(* CoDeSys 2.3.9.13 project: wago_842_1.8.pro *)
(* Libraries: X:\Dev\Wago Calaos\Wago_1.7\DALI_02v2.4.lib 10.3.09 10:32:26, SYSTEM.LIB 6.12.00 08:50:26, Visual.lib 22.2.01 17:57:44, mod_com.lib 17.5.05 08:45:02, Ethernet.lib 8.7.04 10:03:04, Standard.lib 1.12.04 09:59:26 *)

(* PLC configuration (modules and I/O channels)
K-Bus [K_Bus] node 0, in %IB0 out %QB0
Fieldbus variables [FB_VARS] node 1, in %IB512 out %QB512
*)

(* Global variable list: Variables_Globales *)
VAR_GLOBAL
	ConfigDone: BOOL := FALSE; (* Do the config only one time *)
	info : ARRAY[0..63] OF MODULE_INFO; (* I/O Module infos *)

	(* modules infos *)
	nb_module: BYTE;
	nb_module_in: BYTE;
	nb_module_out: BYTE;
	nb_module_analog_in: BYTE;
	nb_module_analog_out: BYTE;
	start_addr_in: WORD;
	start_addr_out: WORD;
	nb_input_digital: WORD;
	nb_output_digital: WORD;

	(* All inputs events *)
	event: ARRAY[0..200] OF INTER_EVENT; (* MAX of 256/8 = 32 digital input modules *)
	lights: ARRAY[0..31] OF BYTE;	(* MAX of 256/8 = 32 digital output modules as lights *)
									(* We store only the boolean state of each light *)
	volets: ARRAY[0..100] OF VOLET; (* MAX of 256/8 = 32 digital output modules as volets *)

	HEARTBEAT: BOOL := FALSE;

	OutArrState: ARRAY[0..512] OF BYTE;	(* state of outputs *)

	impulse_time: TIME := T#300ms;

	(* DALI *)
	DALIJoblist: FbDALI_Joblist;

	Dali_switch: FbDALI_SwitchValue;
	DALIDimmValue: FbDALI_StatusDimmValue;

	byOutArr AT %QB0: ARRAY[0..512] OF BYTE;	(* Byte array in Q memory *)
	byInArr AT %IB0: ARRAY[0..512] OF BYTE;	(* Byte array in I memory *)
END_VAR

(* Data type *)
TYPE OUTPUT_ADDR :
STRUCT

	(* the first ouput address, only needed *)
	ADDR1: BYTE;
	(* the second address used only for the VOLET function bloc *)
	ADDR2: BYTE;

	(* If SameAs <> -1, then a input is wired the same as the specified ID *)
	SameAs: INT := -1;

END_STRUCT
END_TYPE

(* Data type *)
(* Enumerate all type of output.
	NONE: Do nothing.
	TELERUPTEUR: Simulate a telerupteur.
	DIRECT: The input is directly "wired" to the output.
	VOLET: Simulate a volet with one button and 2 output (up and down).
	TELERUPTEUR_DALI: Controls a DALI lamp
	TELERUPTEUR_DALI_GROUP: Controls a DALI group
*)

TYPE OUTPUT_TYPE : (NONE, TELERUPTEUR, DIRECT, VOLET, VOLET_IMPULSE, TELERUPTEUR_DALI, TELERUPTEUR_DALI_GROUP);
END_TYPE

(* Data type *)
(* Enumerate all type of output.
	NONE: Do nothing.
	TELERUPTEUR: Simulate a telerupteur.
	DIRECT: The input is directly "wired" to the output.
	VOLET: Simulate a volet with one button and 2 output (up and down).
*)

TYPE VOLET_MODE : (VOLET_STOP, VOLET_UP, VOLET_DOWN, IMP_UP, IMP_DOWN, IMP_STOP);
END_TYPE

(* POU PLC_PRG, ST *)
PROGRAM PLC_PRG
VAR
	i: INT;
	start: BYTE;
	init_dali: BOOL := FALSE;
END_VAR
(* Main PRG *)

(* Start the config program *)
Config;

IF (Config.CONFIG_DALI = TRUE) THEN

	(* Call DALI jobs to send commands on the DALI bus *)
	DALIJoblist();
	DALI_Config();

	IF (init_dali = FALSE) THEN
		Dali_switch(xButton := FALSE);
		Dali_switch(bAddress := 255, xGroup := FALSE, bDimmLevel := 0,
				         xButton := TRUE);

		init_dali := TRUE;
	END_IF

END_IF


IF (HEARTBEAT = FALSE) THEN
	ManageOutput;
END_IF

(* Read a command from UDP *)
UDPServer;

(* Send inputs status on the network *)
SendInput;

IF (HEARTBEAT = FALSE) THEN
	(* update outputs *)
	FOR i := start_addr_out / 8 TO 512 DO
		byOutArr[i] := OutArrState[i];
	END_FOR
ELSE
	(* update outputs *)
	FOR i := start_addr_out / 8 TO 512 DO
		OutArrState[i] := byOutArr[i];
	END_FOR
END_IF
END_PROGRAM

(* POU Config, ST *)
PROGRAM Config
VAR
	access : MODULE_INFO_ACCESS;
	cpt: BYTE;
	ethernet_config : ETHERNET_SET_VARIABLES;
	CONFIG_DALI: BOOL;

END_VAR
VAR_INPUT RETAIN
	SERVER_IP: DWORD;
	DALI_MODE: BYTE;
END_VAR
VAR CONSTANT
	CALAOS_VERSION_H: WORD := 1;
	CALAOS_VERSION_L: WORD := 8;
	DALI: BYTE := 1;
	DSI: BYTE := 2;
END_VAR
(* Do all the config job *)

IF (ConfigDone = FALSE) THEN

(* Get the module I/O Config *)
access.physicalPosTo := 0;
access.moduleType := 0;
ADD_PI_INFORMATION( 1, ADR(access), ADR(info[0]) );

FOR cpt := 0 TO 63 DO
	IF (info[cpt].moduleType = 0 AND info[cpt].physicalPos = 0) THEN
		cpt := 63; (* the end *)
	ELSE
		IF (info[cpt].moduleType = 641) THEN
			(* This is a DALI module *)
			CONFIG_DALI := TRUE;
		END_IF

		nb_module := nb_module + 1;
		IF ((info[cpt].desc.sizePAE > 8) AND (info[cpt].desc.channels > 0)) THEN
			nb_module_analog_in := nb_module_analog_in + 1;
			start_addr_in := start_addr_in + info[cpt].desc.sizePAE;
		END_IF
		IF ((info[cpt].desc.sizePAA > 8) AND (info[cpt].desc.channels > 0)) THEN
			nb_module_analog_out := nb_module_analog_out + 1;
			start_addr_out := start_addr_out + info[cpt].desc.sizePAA;
		END_IF
		IF ((info[cpt].desc.sizePAE <= 16) AND (info[cpt].desc.sizePAE > 0) AND (info[cpt].desc.channels = 0)) THEN
			nb_module_in := nb_module_in + 1;
			nb_input_digital := nb_input_digital + info[cpt].desc.sizePAE;
		END_IF
		IF ((info[cpt].desc.sizePAA <= 16) AND (info[cpt].desc.sizePAA > 0) AND (info[cpt].desc.channels = 0)) THEN
			nb_module_out := nb_module_out + 1;
			nb_output_digital := nb_output_digital + info[cpt].desc.sizePAA;
		END_IF

	END_IF
END_FOR

(* Start the heartbeat timer *)
(*HEARTBEAT_TIMER(IN:=FALSE, PT:=T#30s);*)
(*HEARTBEAT_TIMER(IN:=TRUE, PT:=T#30s);*)

(* Config du timout des sockets *)
ethernet_config(EN:=TRUE, BootpRequest:=0, ConnectionWdTime:=65535);

ConfigDone := TRUE;

LedInit;
LedStart;

END_IF
END_PROGRAM

(* POU LedInit, ST *)
PROGRAM LedInit
VAR
	Sequence: ARRAY [0..4] OF FLASHING_SEQUENCE;
	ptrFS: POINTER TO FLASHING_SEQUENCE;

END_VAR
Sequence[0].Colour := ORANGE;
Sequence[0].Frequency := 10;
Sequence[0].Relation := 50;
Sequence[0].Duration := t#0s;

Sequence[1].Colour := ORANGE;
Sequence[1].Frequency := 0;
Sequence[1].Relation := 128;
Sequence[1].Duration := t#0s;

Sequence[2].Colour := GREEN;
Sequence[2].Frequency := 0;
Sequence[2].Relation := 128;
Sequence[2].Duration := t#0s;

Sequence[3].Colour := RED;
Sequence[3].Frequency := 0;
Sequence[3].Relation := 128;
Sequence[3].Duration := t#0s;

Sequence[4].Colour := ORANGE;
Sequence[4].Frequency := 0;
Sequence[4].Relation := 0;
Sequence[4].Duration := t#0s;

ptrFS := ADR(Sequence);
SET_FLASHING_SEQUENCE(TRUE, ADR(ptrFS));
END_PROGRAM

(* POU LedStart, ST *)
PROGRAM LedStart
VAR
END_VAR
SET_FLASHING_SEQUENCE_INDEX(TRUE, TRUE, 0);
START_FLASHING_SEQUENCE(TRUE);
END_PROGRAM

(* POU ManageOutput, ST *)
PROGRAM ManageOutput
VAR
	cpt: BYTE;
	tmp: BYTE;
	_light: LIGHT;
END_VAR
VAR_INPUT RETAIN
	output_type: ARRAY[0..256] OF OUTPUT_TYPE; (* The type of each output *)
	output_addr: ARRAY[0..256] OF OUTPUT_ADDR; (* The addresses for each type *)
    	volets_position: ARRAY[0..30] OF DWORD;
END_VAR
(* Set all outputs when in standalone mode *)

(* Get the address of the first digital output *)
FOR cpt := 0 TO UINT_TO_BYTE(nb_input_digital) DO

	CASE output_type[cpt] OF
	NONE: (* Do nothing *);
	TELERUPTEUR:
		tmp := cpt;
		IF (output_addr[cpt].SameAs >= 0) THEN
			tmp := INT_TO_BYTE(output_addr[cpt].SameAs);
		END_IF
		IF (event[cpt].ON = TRUE) THEN
			_light(IN := FALSE, STATE := BYTE_TO_BOOL(SHR(lights[tmp / 8], tmp MOD 8) AND 16#01));
			_light(IN := TRUE, STATE := BYTE_TO_BOOL(SHR(lights[tmp / 8], tmp MOD 8) AND 16#01));
			SetOutput(output_addr[tmp].ADDR1 + start_addr_out, _light.OUT);

			(* set old state *)
			IF (_light.OUT = TRUE) THEN
				lights[tmp / 8] := lights[tmp / 8] OR SHL(16#01, tmp MOD 8);
			ELSE
				lights[tmp / 8] := lights[tmp / 8] AND NOT SHL(16#01, tmp MOD 8);
			END_IF
		END_IF
	DIRECT:
		tmp := cpt;
		IF (output_addr[cpt].SameAs >= 0) THEN
			tmp := INT_TO_BYTE(output_addr[cpt].SameAs);
		END_IF
		SetOutput(output_addr[tmp].ADDR1 + start_addr_out, GetInput(cpt + start_addr_in));
	VOLET:
		tmp := cpt;
		IF (output_addr[cpt].SameAs >= 0) THEN
			tmp := INT_TO_BYTE(output_addr[cpt].SameAs);
		END_IF
		IF (event[cpt].ON = TRUE) THEN
			volets[tmp](IN := TRUE, IMPULSE := FALSE);
			SetOutput(output_addr[tmp].ADDR1 + start_addr_out, volets[tmp].MONTE);
			SetOutput(output_addr[tmp].ADDR2 + start_addr_out, volets[tmp].DESCENTE);
		END_IF
	VOLET_IMPULSE:
		tmp := cpt;
		IF (output_addr[cpt].SameAs >= 0) THEN
			tmp := INT_TO_BYTE(output_addr[cpt].SameAs);
		END_IF
		IF (event[cpt].ON = TRUE) THEN
			volets[tmp](IN := TRUE, IMPULSE := TRUE);
		ELSE
			volets[tmp](IN := FALSE, IMPULSE := TRUE);
		END_IF
		SetOutput(output_addr[tmp].ADDR1 + start_addr_out, volets[tmp].MONTE);
		SetOutput(output_addr[tmp].ADDR2 + start_addr_out, volets[tmp].DESCENTE);
	TELERUPTEUR_DALI:
		tmp := cpt;
		IF (output_addr[cpt].SameAs >= 0) THEN
			tmp := INT_TO_BYTE(output_addr[cpt].SameAs);
		END_IF
		IF (event[cpt].ON = TRUE) THEN
			_light(IN := FALSE, STATE := BYTE_TO_BOOL(SHR(lights[tmp / 8], tmp MOD 8) AND 16#01));
			_light(IN := TRUE, STATE := BYTE_TO_BOOL(SHR(lights[tmp / 8], tmp MOD 8) AND 16#01));

			Dali_switch(xButton := FALSE);
			IF (_light.OUT = TRUE) THEN
				Dali_switch(bAddress := output_addr[tmp].ADDR2, xGroup := FALSE, bDimmLevel := 100,
					bFadeTime := 1, xButton := TRUE);
			ELSE
				Dali_switch(bAddress := output_addr[tmp].ADDR2, xGroup := FALSE, bDimmLevel := 0,
					bFadeTime := 1, xButton := TRUE);
			END_IF

			(* set old state *)
			IF (_light.OUT = TRUE) THEN
				lights[tmp / 8] := lights[tmp / 8] OR SHL(16#01, tmp MOD 8);
			ELSE
				lights[tmp / 8] := lights[tmp / 8] AND NOT SHL(16#01, tmp MOD 8);
			END_IF
		END_IF
	TELERUPTEUR_DALI_GROUP:
		tmp := cpt;
		IF (output_addr[cpt].SameAs >= 0) THEN
			tmp := INT_TO_BYTE(output_addr[cpt].SameAs);
		END_IF
		IF (event[cpt].ON = TRUE) THEN
			_light(IN := FALSE, STATE := BYTE_TO_BOOL(SHR(lights[tmp / 8], tmp MOD 8) AND 16#01));
			_light(IN := TRUE, STATE := BYTE_TO_BOOL(SHR(lights[tmp / 8], tmp MOD 8) AND 16#01));
			Dali_switch(xButton := FALSE);
			IF (_light.OUT = TRUE) THEN
				Dali_switch(bAddress := output_addr[tmp].ADDR2, xGroup := TRUE, bDimmLevel := 100,
					bFadeTime := 1, xButton := TRUE);
			ELSE
				Dali_switch(bAddress := output_addr[tmp].ADDR2, xGroup := TRUE, bDimmLevel := 0,
					bFadeTime := 1, xButton := TRUE);
			END_IF

			(* set old state *)
			IF (_light.OUT = TRUE) THEN
				lights[tmp / 8] := lights[tmp / 8] OR SHL(16#01, tmp MOD 8);
			ELSE
				lights[tmp / 8] := lights[tmp / 8] AND NOT SHL(16#01, tmp MOD 8);
			END_IF
		END_IF
	END_CASE
END_FOR
END_PROGRAM

(* POU LIGHT, ST *)
FUNCTION_BLOCK LIGHT
VAR
	TRIG: R_TRIG;
	light: BOOL;
END_VAR
VAR_INPUT
	IN: BOOL;
	STATE: BOOL;
END_VAR
VAR_OUTPUT
	OUT: BOOL;
END_VAR
(* telerupteur *)

TRIG(CLK := IN);
light := TRIG.Q;

OUT := STATE;

IF light = TRUE THEN
	IF OUT = TRUE THEN
		OUT := FALSE;
	ELSE
		OUT := TRUE;
	END_IF;
END_IF;
END_FUNCTION_BLOCK

(* POU SetOutput, ST *)
FUNCTION SetOutput : BOOL
VAR_INPUT
	bit_offset: UINT;
	val: BOOL;
END_VAR
VAR
END_VAR
(* get the byte AND  select the bit *)

(* Take care of special modules *
bit_offset := bit_offset + start_addr_out; *)

IF (HEARTBEAT = FALSE) THEN
	IF (val = TRUE) THEN
		OutArrState[bit_offset / 8] := OutArrState[bit_offset / 8] OR SHL(16#01, bit_offset MOD 8);
	ELSE
		OutArrState[bit_offset / 8] := OutArrState[bit_offset / 8] AND NOT SHL(16#01, bit_offset MOD 8);
	END_IF

ELSE
	IF (val = TRUE) THEN
		byOutArr[bit_offset / 8] := byOutArr[bit_offset / 8] OR SHL(16#01, bit_offset MOD 8);
	ELSE
		byOutArr[bit_offset / 8] := byOutArr[bit_offset / 8] AND NOT SHL(16#01, bit_offset MOD 8);
	END_IF
END_IF

SetOutput := TRUE;
END_FUNCTION

(* POU GetInput, ST *)
FUNCTION GetInput : BOOL
VAR_INPUT
	bit_offset: UINT;
END_VAR
VAR
END_VAR
VAR CONSTANT
	byBitArr: ARRAY[0..7] OF BYTE := 16#01,16#02,16#04,16#08,16#10,16#20,16#40,16#80;
END_VAR
(* get the byte AND  select the bit *)

GetInput := BYTE_TO_BOOL(byInArr[bit_offset/8] AND byBitArr[bit_offset MOD 8]);
END_FUNCTION

(* POU VOLET, ST *)
FUNCTION_BLOCK VOLET
VAR
	sens: BOOL;
	imp: TP;
	mode: VOLET_MODE;
END_VAR
VAR_INPUT
	IN: BOOL;
	IMPULSE: BOOL;
END_VAR
VAR_OUTPUT
	MONTE: BOOL;
	DESCENTE:BOOL;
END_VAR
(* Volet *)

IF IMPULSE = FALSE THEN
	(* Normal mode *)
	IF (MONTE = TRUE OR DESCENTE = TRUE) THEN
		MONTE := FALSE;
		DESCENTE := FALSE;
	ELSE

		IF IN = TRUE THEN
			IF sens = TRUE THEN
				sens := FALSE;
			ELSE
				sens := TRUE;
			END_IF;

			IF sens = TRUE THEN
				(*monte*)
				DESCENTE := FALSE;
				MONTE := TRUE;
			ELSE
				MONTE := FALSE;
				DESCENTE := TRUE;
			END_IF;
		END_IF

	END_IF
ELSE
	(* impulse mode *)
	imp(IN := FALSE, PT:= impulse_time);

	IF mode = IMP_STOP THEN
		MONTE := imp.Q;
		DESCENTE := imp.Q;
		IF imp.Q = FALSE THEN
			mode := VOLET_STOP;
		END_IF;
	END_IF;
	IF mode = IMP_UP THEN
		MONTE := imp.Q;
		DESCENTE := FALSE;
		IF imp.Q = FALSE THEN
			mode := VOLET_UP;
		END_IF;
	END_IF;
	IF mode = IMP_DOWN THEN
		MONTE := FALSE;
		DESCENTE := imp.Q;
		IF imp.Q = FALSE THEN
			mode := VOLET_DOWN;
		END_IF;
	END_IF;

	IF mode = VOLET_UP OR mode = VOLET_DOWN THEN
		IF IN = TRUE THEN
			imp(IN := TRUE, PT:= impulse_time);
			mode := IMP_STOP;
		END_IF;
	ELSE
		IF IN = TRUE THEN
			IF sens = TRUE THEN
				sens := FALSE;
			ELSE
				sens := TRUE;
			END_IF;

			IF sens = TRUE THEN
				imp(IN := TRUE, PT:= impulse_time);
				mode := IMP_UP;
			ELSE
				imp(IN := TRUE, PT:= impulse_time);
				mode := IMP_DOWN;
			END_IF;
		END_IF;
	END_IF;
END_IF;
END_FUNCTION_BLOCK

(* POU UDPServer, ST *)
PROGRAM UDPServer
VAR
	server: EthernetServer_FB;

	rBuffer, wBuffer: POINTER TO BYTE;
	buffer: ARRAY[1 .. 1500] OF BYTE;
	cmd: STRING(255);
	start_send: BOOL := FALSE;
	i: WORD;
	dali_group: BOOL;

	HEARTBEAT_TIMER: TON;

	p1: DINT;
	p2: DINT;
	p3: DINT;
	p4: DINT;
	p5: DINT;
	ip1, ip2, ip3, ip4: DWORD;
	DaliSend: BOOL := FALSE;

	(* Used by dali config for answer
	   0 = no action
	   1 = Search all active address
	   2 = Read groups for short adress
	*)
	DaliSendAction: BYTE := 0;

(*	DALIShowShortAdr: FbDALI_ShowShortAdr;
	DALIConfigDevice: FbDALI_ConfigDevice;*)

END_VAR
(* Here we start an UDP server for other network functions *)

HEARTBEAT_TIMER(IN:=TRUE, PT:=T#30s);

rBuffer := ADR(buffer);
wBuffer := ADR(cmd);

cmd := CONCAT(cmd, ASCIIBYTE_TO_STRING(0));

server.tTIMEOUT	:= t#60s;
server.xTCP_PROTOCOL := FALSE;
server.wPORT := 4646;
server.iBYTES_TO_SEND := LEN(cmd) + 1;
server(xOPEN_SERVER := TRUE, xSTART_SEND := start_send, ptSEND_BUFFER := wBuffer, ptRECV_BUFFER := rBuffer);

IF server.bDataReceived THEN

	cmd := '';
	FOR i := 1 TO server.iBYTES_RECEIVED DO
		cmd := CONCAT(cmd, ASCIIBYTE_TO_STRING(buffer[i]));
	END_FOR

	IF (STRING_COMPARE(cmd, 'WAGO_HEARTBEAT') = TRUE) THEN
		HEARTBEAT_TIMER(IN:=FALSE, PT:=T#30s);
		HEARTBEAT_TIMER(IN:=TRUE, PT:=T#30s);

		LedModePC;
	END_IF

	IF (Strncmp(cmd, 'WAGO_SET_OUTTYPE ', 17) = TRUE) THEN
		p1 := GET_PARAM_DINT(cmd, 1);
		p2 := GET_PARAM_DINT(cmd, 2);
		CASE p2 OF
		0: ManageOutput.output_type[p1] := NONE;
		1: ManageOutput.output_type[p1] := TELERUPTEUR;
		2: ManageOutput.output_type[p1] := DIRECT;
		3: ManageOutput.output_type[p1] := VOLET;
		4: ManageOutput.output_type[p1] := VOLET_IMPULSE;
		5: ManageOutput.output_type[p1] := TELERUPTEUR_DALI;
		6: ManageOutput.output_type[p1] := TELERUPTEUR_DALI_GROUP;
		END_CASE
	END_IF

	IF (Strncmp(cmd, 'WAGO_SET_OUTADDR ', 17) = TRUE) THEN
		p1 := GET_PARAM_DINT(cmd, 1);
		p2 := GET_PARAM_DINT(cmd, 2);
		p3 := GET_PARAM_DINT(cmd, 3);
		p4 := GET_PARAM_DINT(cmd, 4);
		ManageOutput.output_addr[p1].ADDR1 := DINT_TO_BYTE(p2);
		ManageOutput.output_addr[p1].ADDR2 := DINT_TO_BYTE(p3);
		ManageOutput.output_addr[p1].SameAs := DINT_TO_INT(p4);
	END_IF

	IF (Strncmp(cmd, 'WAGO_GET_OUTTYPE ', 17) = TRUE) THEN
		p1 := GET_PARAM_DINT(cmd, 1);
		cmd := 'WAGO_OUTTYPE ';
		cmd := CONCAT(cmd, ITOA(DINT_TO_INT(p1)));
		cmd := CONCAT(cmd, ' ');
		CASE ManageOutput.output_type[p1] OF
		NONE: cmd := CONCAT(cmd, ITOA(0));;
		TELERUPTEUR: cmd := CONCAT(cmd, ITOA(1));;
		DIRECT: cmd := CONCAT(cmd, ITOA(2));;
		VOLET: cmd := CONCAT(cmd, ITOA(3));;
		VOLET_IMPULSE: cmd := CONCAT(cmd, ITOA(4));;
		TELERUPTEUR_DALI: cmd := CONCAT(cmd, ITOA(5));;
		TELERUPTEUR_DALI_GROUP: cmd := CONCAT(cmd, ITOA(6));;
		END_CASE
		start_send := TRUE;
	END_IF

	IF (Strncmp(cmd, 'WAGO_GET_OUTADDR ', 17) = TRUE) THEN
		p1 := GET_PARAM_DINT(cmd, 1);
		cmd := 'WAGO_OUTADDR ';
		cmd := CONCAT(cmd, ITOA(DINT_TO_INT(p1)));
		cmd := CONCAT(cmd, ' ');
		cmd := CONCAT(cmd, ITOA(ManageOutput.output_addr[p1].ADDR1));
		cmd := CONCAT(cmd, ' ');
		cmd := CONCAT(cmd, ITOA(ManageOutput.output_addr[p1].ADDR2));
		cmd := CONCAT(cmd, ' ');
		cmd := CONCAT(cmd, ITOA(ManageOutput.output_addr[p1].SameAs));
		start_send := TRUE;
	END_IF

	IF (STRING_COMPARE(cmd, 'WAGO_GET_INFO') = TRUE) THEN
		cmd := 'WAGO_INFO ';
		cmd := CONCAT(cmd, ITOA(nb_module));
		cmd := CONCAT(cmd, ' ');
		cmd := CONCAT(cmd, ITOA(nb_module_in));
		cmd := CONCAT(cmd, ' ');
		cmd := CONCAT(cmd, ITOA(WORD_TO_INT(nb_module_out)));
		cmd := CONCAT(cmd, ' ');
		cmd := CONCAT(cmd, ITOA(WORD_TO_INT(nb_input_digital)));
		cmd := CONCAT(cmd, ' ');
		cmd := CONCAT(cmd, ITOA(WORD_TO_INT(nb_output_digital)));
		cmd := CONCAT(cmd, ' ');
		cmd := CONCAT(cmd, ITOA(nb_module_analog_in));
		cmd := CONCAT(cmd, ' ');
		cmd := CONCAT(cmd, ITOA(nb_module_analog_out));
		start_send := TRUE;
	END_IF

	IF (Strncmp(cmd, 'WAGO_GET_INFO_MODULE ', 21) = TRUE) THEN
		p1 := GET_PARAM_DINT(cmd, 1);
		cmd := 'WAGO_MODULE ';
		cmd := CONCAT(cmd, ITOA(DINT_TO_INT(p1)));
		cmd := CONCAT(cmd, ' ');
		cmd := CONCAT(cmd, ITOA(WORD_TO_INT(info[p1].moduleType)));
		cmd := CONCAT(cmd, ' ');
		cmd := CONCAT(cmd, ITOA(info[p1].physicalPos));
		cmd := CONCAT(cmd, ' ');
		cmd := CONCAT(cmd, ITOA(info[p1].desc.sizePAE));
		cmd := CONCAT(cmd, ' ');
		cmd := CONCAT(cmd, ITOA(info[p1].desc.sizePAA));
		start_send := TRUE;
	END_IF

	IF (Strncmp(cmd, 'WAGO_SET_SERVER_IP ', 19) = TRUE) THEN
		cmd := DELETE(cmd, 19, 1);
		(* deletes the dot  *)
		cmd := REPLACE(cmd, ' ', 1, FIND(cmd, '.'));
		cmd := REPLACE(cmd, ' ', 1, FIND(cmd, '.'));
		cmd := REPLACE(cmd, ' ', 1, FIND(cmd, '.'));
		ip1 := GET_PARAM_DINT(cmd, 0);
		ip2 := GET_PARAM_DINT(cmd, 1);
		ip3 := GET_PARAM_DINT(cmd, 2);
		ip4 := GET_PARAM_DINT(cmd, 3);
		Config.SERVER_IP := SHL(ip1, 24) OR SHL(ip2, 16) OR SHL(ip3, 8) OR ip4;
	END_IF

	IF (Strncmp(cmd, 'WAGO_SET_OUTPUT ', 16) = TRUE) THEN
		p1 := GET_PARAM_DINT(cmd, 1);
		p2 := GET_PARAM_DINT(cmd, 2);

		p1 := start_addr_out + p1;

		IF (p2 = 1) THEN
			SetOutput(DINT_TO_UINT(p1), TRUE);
		ELSE
			SetOutput(DINT_TO_UINT(p1), FALSE);
		END_IF
	END_IF

	IF (Strncmp(cmd, 'WAGO_GET_VERSION', 16) = TRUE) THEN
		cmd := 'WAGO_GET_VERSION ';
		cmd := CONCAT(cmd, ITOA(WORD_TO_INT(Config.CALAOS_VERSION_H)));
		cmd := CONCAT(cmd, '.');
		cmd := CONCAT(cmd, ITOA(WORD_TO_INT(Config.CALAOS_VERSION_L)));
		start_send := TRUE;
	END_IF

	IF (Strncmp(cmd, 'WAGO_DALI_SET ', 14) = TRUE) THEN
		p1 := GET_PARAM_DINT(cmd, 1); (* Dali Line *)
		p2 := GET_PARAM_DINT(cmd, 2); (* Short addr or group? *)
		p3 := GET_PARAM_DINT(cmd, 3); (* Dali Address *)
		p4 := GET_PARAM_DINT(cmd, 4); (* Dimm value in percent *)
		p5 := GET_PARAM_DINT(cmd, 5); (* Fade time *)

		IF (p2 = 1) THEN
			dali_group := TRUE;
		ELSE
			dali_group := FALSE;
		END_IF

		Dali_switch(xButton := FALSE);
		Dali_switch(bAddress := DINT_TO_BYTE(p3), xGroup := dali_group, bDimmLevel := DINT_TO_BYTE(p4),
			bFadeTime := DINT_TO_BYTE(p5), xButton := TRUE);
	END_IF

	IF (Strncmp(cmd, 'WAGO_DALI_GET ', 14) = TRUE) THEN
		p1 := GET_PARAM_DINT(cmd, 1); (* Dali Line *)
		p2 := GET_PARAM_DINT(cmd, 2); (* Short addr *)
		p3 := GET_PARAM_DINT(cmd, 3); (* Dali Address *)
		p4 := GET_PARAM_DINT(cmd, 4); (* Dimm value in percent *)
		p5 := GET_PARAM_DINT(cmd, 5); (* Fade time *)

		IF (p2 = 1) THEN
			dali_group := TRUE;
		ELSE
			dali_group := FALSE;
		END_IF

		DALIDimmValue(xEnable := TRUE, bShortAddress := DINT_TO_BYTE(p2), tCycleTime := t#1s);
		DaliSend := TRUE;
	END_IF

    IF (Strncmp(cmd, 'WAGO_INFO_VOLET_GET ', 20) = TRUE) THEN
		p1 := GET_PARAM_DINT(cmd, 1);
		cmd := 'WAGO_INFO_VOLET ';
		cmd := CONCAT(cmd, ITOA(DINT_TO_INT(p1)));
		cmd := CONCAT(cmd, ' ');
(*		cmd := CONCAT(cmd, ITOA(DWORD_TO_INT(ManageOutput.volets_position[p1]))); *)
		cmd := CONCAT(cmd, DWORD_TO_STRING(ManageOutput.volets_position[p1]));
		start_send := TRUE;
	END_IF

    IF (Strncmp(cmd, 'WAGO_INFO_VOLET_SET ', 20) = TRUE) THEN
		p1 := GET_PARAM_DINT(cmd, 1);
		p2 := GET_PARAM_DINT(cmd, 2);
		ManageOutput.volets_position[p1] := DINT_TO_DWORD(p2);
	END_IF
END_IF

IF (DaliSend = TRUE) THEN
	IF (DALIDimmValue.xReady = TRUE) THEN
		cmd := 'WAGO_DALI_GET ';
		cmd := CONCAT(cmd, ITOA(BOOL_TO_INT(DALIDimmValue.xStatus)));
		cmd := CONCAT(cmd, ' ');
		cmd := CONCAT(cmd, ITOA(BYTE_TO_INT(DALIDimmValue.bDimmValue)));
		start_send := TRUE;
		DaliSend := FALSE;
	ELSE
		DALIDimmValue(xEnable := TRUE, bShortAddress := DINT_TO_BYTE(p2), tCycleTime := t#1s);
	END_IF;
END_IF

IF (HEARTBEAT_TIMER.Q = TRUE) THEN
	(* We lost the connection with the server *)
	(* The wago is now in standalone mode *)
	HEARTBEAT := FALSE;

	LedModeWAGO;
ELSE
	HEARTBEAT := TRUE;
END_IF
END_PROGRAM

(* POU EthernetServer_FB, ST *)
FUNCTION_BLOCK EthernetServer_FB
(************************************************************)
(* ETHERNET_SERVER		                          		    *)
(* Ver. 1.0   	                                         	*)
(* Date:  10.02.2003					         	 		*)
(* Author:  Volker Begemann                            		*)
(************************************************************)
VAR_INPUT
	xOPEN_SERVER		:	BOOL;				(* Set TRUE to enable function block			*)
	wPORT					:	WORD;				(* Port number											*)
	xTCP_PROTOCOL		:	BOOL;				(* TRUE => TCP; FALSE => UDP						*)
	tTIMEOUT				:	TIME:=t#20s;	(* Watchdog timeout value (seconds)				*)
	iBYTES_TO_SEND		:	INT;				(* Number of bytes to transmit					*)
	ptSEND_BUFFER		:	POINTER TO ARRAY[1..1500] OF BYTE;		(* Transmit Buffer	*)
END_VAR
VAR_IN_OUT
	xSTART_SEND:		BOOL;						(* Set TRUE to initiate data transmittal, will be	*)
														(* reset FALSE when transmittal is completed 		*)
(* 	utRECEIVE_BUFFER:	typEthernetBuffer;	(* Receive Buffer *) *)
	ptRECV_BUFFER		:	POINTER TO ARRAY[1..1500] OF BYTE;		(* Receive Buffer	*)
END_VAR
VAR_OUTPUT
	utERROR					:	ETH_ERROR;	(* See ETH_ERROR datatype in ETHERNET.LIB	*)
													(* for error codes and definitions			*)
	xSERVER_OPEN:			BOOL;				(* TRUE if socket connection made			*)
	wSOCKET:					WORD;				(* Socket connection number					*)
	bDataReceived: 		BOOL := FALSE;
	iBYTES_RECEIVED: INT; (* Number of bytes received *)
END_VAR
VAR
	i: INT;
	CloseState:			INT;
	EthernetOpen:		ETHERNET_SERVER_OPEN;
	EthernetClose:		ETHERNET_SERVER_CLOSE;
	EthernetWrite:		ETHERNET_WRITE;
	EthernetRead:		ETHERNET_READ;
	GetConfig:			ETHERNET_GET_NETWORK_CONFIG;
	EthernetBuffer:	ARRAY[1..1500] OF BYTE;
	Status:				WORD:=0;
	client_SRC_PORT:	WORD;
	watchdog_timer1:	TON;
	client_SRC_IP:		DWORD;
END_VAR
IF xOPEN_SERVER THEN
	watchdog_timer1(IN:=TRUE , PT:=tTIMEOUT );

	IF watchdog_timer1.q THEN
		watchdog_timer1(IN:=FALSE , PT:=tTIMEOUT );
		EthernetClose(EN:= 1, SOCKET:= EthernetOpen.SOCKET);
		EthernetClose(EN:= 0, SOCKET:= 0);
		Status := 0; (* Try to open the server *)
	END_IF

	CASE Status OF
		0:
			GetConfig(EN:=FALSE );
			GetConfig(EN:=TRUE );
			utERROR		:=	0;
			wSocket		:=	0;
			CloseState	:=	0;
			status		:=	1;
		1:
			GetConfig(EN:=TRUE );
			IF GetConfig.ENO THEN
				IF GetConfig.IP_ADR<>0 THEN
					status:=4;
					EthernetOpen (EN:=0);
					EthernetRead(EN:= 0, SOCKET:=0 ,  DATA:=EthernetBuffer );
					EthernetClose(EN:= 0);
				ELSE
					status:=0;
				END_IF
			END_IF
		4: 	(* try to open a socket*)
			IF xTCP_PROTOCOL THEN
				EthernetOpen(EN:=1 , TYP:=SOCK_STREAM, PROTO := IPPROTO_TCP, PORT := wPort);
			ELSE
				EthernetOpen(EN:=1 , TYP:=SOCK_DGRAM, PROTO := IPPROTO_UDP, PORT := wPort);
			END_IF
			IF ((EthernetOpen.ERROR = 0) AND (EthernetOpen.ENO = 1)) THEN
				Status  := 10; (* socket created, wait for data to process *)
				EthernetOpen (EN:=0);
				xServer_open:=TRUE;
				wSocket:=EthernetOpen.socket;
			ELSE
				Status := 0; 	(* socket not available, try it again *)
				EthernetOpen (EN:=0);
				xServer_open:=FALSE;
				wSocket:=0;
			END_IF;

		10: 	(* Wait for data to process *)
			(* Monitor ethernet port for new data *)
			bDataReceived	:= FALSE;
	 		EthernetRead(	EN:= 1, SOCKET:=EthernetOpen.SOCKET, DATA:=EthernetBuffer);
			EthernetRead(	EN:= 0, SOCKET:=0, DATA:=EthernetBuffer);

			IF(EthernetRead.ERROR<>0) THEN  			(* Error reading the socket, close it *)
				Status	:=	40;
			ELSIF (EthernetRead.LEN_OUT <>0) THEN  (* Process the data received via the ethernet port *)
				client_SRC_IP		:=	EthernetRead.SRC_IP;
				client_SRC_PORT	:=	EthernetRead.SRC_PORT;
				ptRECV_BUFFER^		:= EthernetBuffer;
				bDataReceived		:= TRUE;
				iBYTES_RECEIVED		:= EthernetRead.LEN_OUT;
				watchdog_timer1(IN:=FALSE, PT:=tTIMEOUT );
			ELSIF (iBytes_TO_SEND > 0 AND xSTART_SEND) THEN  (* Process the data received *)
				EthernetWrite(EN:= 0, DATA:=EthernetBuffer);
				status	:=	30;
			END_IF

		30: 	(* Process the data to send *)
			EthernetBuffer :=ptSEND_BUFFER^;
			(* Send data in transmit buffer out ethernet port *)
			IF xTCP_PROTOCOL THEN
					EthernetWrite(	EN:= 1,
								SOCKET:= EthernetOpen.SOCKET,
								LEN_IN:=iBYTES_TO_SEND,
								DATA:=EthernetBuffer );
			ELSE
				IF client_SRC_IP>0 AND client_SRC_PORT>0 THEN
					EthernetWrite(EN:=1, SOCKET:=EthernetOpen.SOCKET , LEN_IN:=iBYTES_TO_SENd , DST_IP:=client_SRC_IP,DST_PORT:=client_SRC_PORT,DATA:=EthernetBuffer );
				ELSE
					status:=10;
				END_IF
			END_IF

			IF EthernetWrite.eno THEN
				IF(EthernetWrite.ERROR <>0) THEN
					Status:=40;(* Error writing to the socket, close it *)
				ELSE
					Status:=10; (* Comms complete, read more data *)
				END_IF;
				xStart_send:=FALSE;
			END_IF
		40:	(* Close the server *)
			EthernetClose(EN:= 1, SOCKET:= EthernetOpen.SOCKET);
			IF EthernetClose.eno THEN
				EthernetClose(EN:= 0);
				xOPEN_SERVER:=FALSE;
				utERROR:=0;
				wSocket:=0;
				Status := 0; (* Try to open the server again *)
			END_IF

	END_CASE;
ELSE
	CASE CloseState OF
	0:
		EthernetClose(EN:= 0);
		EthernetClose(EN:= 1, SOCKET:= EthernetOpen.SOCKET);
		CloseState:=1;
	1:
		EthernetClose(EN:= 1, SOCKET:= EthernetOpen.SOCKET);
		IF EthernetClose.eno THEN
			EthernetClose(EN:= 0);
			CloseState:=2;
		END_IF
	2:
		xOPEN_SERVER:=FALSE;
		utERROR:=0;
		wSocket:=0;
	END_CASE
END_IF
END_FUNCTION_BLOCK

(* POU LedModePC, ST *)
PROGRAM LedModePC
VAR
END_VAR
SET_FLASHING_SEQUENCE_INDEX(TRUE, TRUE, 2);
END_PROGRAM

(* POU Strncmp, ST *)
FUNCTION Strncmp : BOOL
VAR_INPUT
	str1: STRING;
	str2: STRING;
	n: BYTE;
END_VAR
VAR
	tmp1: POINTER TO ARRAY[0..255] OF BYTE;
	tmp2: POINTER TO ARRAY[0..255] OF BYTE;
	i: BYTE;
END_VAR
tmp1 := ADR(str1);
tmp2 := ADR(str2);

Strncmp := TRUE;

FOR i := 0 TO n - 1 DO
	IF (tmp1^[i] <> tmp2^[i]) THEN
		Strncmp := FALSE;
		i := n;
	END_IF
END_FOR
END_FUNCTION

(* POU GET_PARAM_DINT, ST *)
FUNCTION GET_PARAM_DINT : DINT
VAR_INPUT
	str: STRING;
	pos: BYTE;
END_VAR
VAR
	i: BYTE;
	j: BYTE;
	mult : DWORD;
	dec : DWORD;
	p: INT;
	tmp: POINTER TO ARRAY[0..255] OF BYTE;
	val: DINT;
	neg: BOOL := FALSE;
END_VAR
(* cut before the value we want *)
FOR i := 1 TO pos DO
	str := DELETE(str, FIND(str, ' '), 1);
END_FOR

(* cut after the value we want *)
p := FIND(str, ' ');
IF (p > 0) THEN
	str := LEFT(str, p - 1);
END_IF

(* Convert the value *)
tmp := ADR(str);

IF (Strncmp(str, '-', 1) = TRUE) THEN
	neg := TRUE;
	str := DELETE(str, 1, 1);
END_IF

val := 0;
FOR i := 0 TO INT_TO_BYTE(LEN(str) - 1) DO
	dec := 1;
	FOR j := 2 TO INT_TO_BYTE(LEN(str) - i) DO
		dec := dec * 10;
	END_FOR

	mult := tmp^[i] - 16#30;
	mult := mult * dec;
	val := val + mult;

END_FOR

(*
CASE LEN(str) OF
	1: val := tmp^[0] - 16#30;
	2: val := (tmp^[0] - 16#30) * 10 + tmp^[1] - 16#30;
	3: val := (tmp^[0] - 16#30) * 100 + (tmp^[1] - 16#30) * 10 + tmp^[2] - 16#30;
END_CASE
*)

IF (neg = TRUE) THEN
	GET_PARAM_DINT := 0 - val;
ELSE
	GET_PARAM_DINT := val;
END_IF
END_FUNCTION

(* POU ITOA, ST *)
FUNCTION ITOA : STRING
VAR_INPUT
	VAL: INT;
END_VAR
VAR
	tmp: INT;
	conv: INT;
END_VAR
(* Convert a byte to string *)

IF (VAL < 0) THEN
	tmp := -VAL;
ELSE
	tmp := VAL;
END_IF

IF (tmp = 0) THEN
	ITOA := ASCIIBYTE_TO_STRING(0 + 16#30);
END_IF

WHILE (tmp > 0) DO
	conv := tmp MOD 10;
	tmp := tmp / 10;
	ITOA := INSERT(ITOA, ASCIIBYTE_TO_STRING(INT_TO_BYTE(conv) + 16#30), 0);
END_WHILE

IF (VAL < 0) THEN
	ITOA := INSERT(ITOA, '-', 0);
END_IF
END_FUNCTION

(* POU LedModeWAGO, ST *)
PROGRAM LedModeWAGO
VAR
END_VAR
SET_FLASHING_SEQUENCE_INDEX(TRUE, TRUE, 1);
END_PROGRAM

(* POU SendInput, ST *)
PROGRAM SendInput
VAR
	cpt: BYTE;
END_VAR
(* Get all inputs *)

(* Get the address of the first digital input *)
FOR cpt := 0 TO UINT_TO_BYTE(nb_input_digital) DO
	event[cpt](IN := GetInput(cpt + start_addr_in));
(*	IF (HEARTBEAT = TRUE) THEN *)
		IF (event[cpt].ON = TRUE) THEN
			SOCK_SEND(cpt, TRUE);
		END_IF
		IF (event[cpt].OFF = TRUE) THEN
			SOCK_SEND(cpt, FALSE);
		END_IF
(*	END_IF *)
END_FOR
END_PROGRAM

(* POU SOCK_SEND, ST *)
FUNCTION SOCK_SEND : BOOL
VAR_INPUT
	num_id: BYTE;
	on: BOOL;
END_VAR
VAR
	socket: ETHERNET_CLIENT_OPEN;
	Close: ETHERNET_CLIENT_CLOSE;
	Write: ETHERNET_WRITE_PT;
	str: STRING(15);
	buffer: POINTER TO ARRAY[1..1500] OF BYTE;
END_VAR
(* Create an UDP socket *)

socket(EN:=0);
socket(EN:=1 , TYP:=SOCK_DGRAM, PROTO:=IPPROTO_UDP , IP_ADR:=0 , PORT:=0);

IF ((socket.ERROR = NO_ERROR) AND (socket.ENO = TRUE)) THEN
	str := 'WAGO INT ';
	str := CONCAT(str,  ITOA(num_id));
	IF (on = TRUE) THEN
		str := CONCAT(str,  ' 1');
	ELSE
		str := CONCAT(str,  ' 0');
	END_IF

	buffer := ADR(str);

	(* send an udp packet *)
	Write(EN:=1, SOCKET:=socket.SOCKET, LEN_IN:=LEN(str), DST_IP:=Config.SERVER_IP, DST_PORT:=4646, DATA_PT:=buffer);
	Write(EN:=0, SOCKET:=0, LEN_IN:=0, DST_IP:=0, DST_PORT:=0, DATA_PT:=buffer);

	IF(Write.ERROR <> NO_ERROR) THEN
		SOCK_SEND := FALSE;
	ELSE
		SOCK_SEND := TRUE;
	END_IF;

	(* Close socket *)
	Close(EN:=1, SOCKET:=socket.SOCKET);
	Close(EN:=0, SOCKET:=0);

ELSE
	SOCK_SEND := FALSE;
END_IF
END_FUNCTION

(* POU LedError, ST *)
PROGRAM LedError
VAR
END_VAR
SET_FLASHING_SEQUENCE_INDEX(TRUE, TRUE, 3);
END_PROGRAM

(* POU INTER_EVENT, ST *)
FUNCTION_BLOCK INTER_EVENT
VAR_INPUT
	IN: BOOL;
END_VAR
VAR_OUTPUT
	ON: BOOL;
	OFF: BOOL;
END_VAR
VAR
	MTRIG: R_TRIG;
	DTRIG: F_TRIG;
END_VAR
(* Get the ON or OFF event on an input *)

MTRIG(CLK := IN);
ON := MTRIG.Q;
DTRIG(CLK := IN);
OFF := DTRIG.Q;
END_FUNCTION_BLOCK

(* Visualisation Addressing
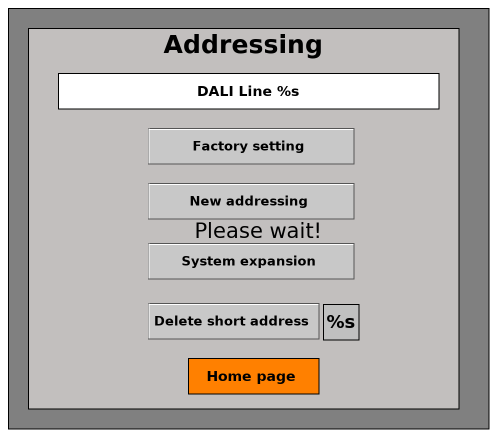
rectangle at (185,80)-(616,461): text "Addressing"
button at (305,235)-(511,271): text "New addressing"; taps DALI_Config.NewAddress; tooltip You have to click and hold the button "New Addressing" longer than two seconds to start the new addressing.
button at (305,295)-(511,331): text "System expansion"; taps DALI_Config.xErweitert; tooltip If you click the button "System expansion", only the ECGs with no short address will be addressed.
rectangle at (480,356)-(516,392): text "%s"; shows DALI_Config.LoeschKurzadr; tooltip Enter the short address to be deleted (1 - 64).; editable
rounded rectangle at (345,410)-(476,446): text "Home page"; opens PLC_VISU; tooltip Back to home page
button at (305,180)-(511,216): text "Factory setting"; taps DALI_Config.Reset; tooltip To reset the ECG you have to click and hold the button two seconds. Group and scene configurations will be deleted.
button at (305,355)-(476,391): text "Delete short address"; taps DALI_Config.Loeschen; tooltip The selected short address will be deleted.
rectangle at (275,97)-(556,468): text "Please wait!"; invisible if not DALI_Config.JobMerker[5]
rounded rectangle at (215,125)-(596,161): text "DALI Line %s"; shows DALI_Config.bDali_Linie; tooltip You can change the DALI Line only on the home page.
1 more shapes without text or variables
*)

(* Visualisation ECG_settings
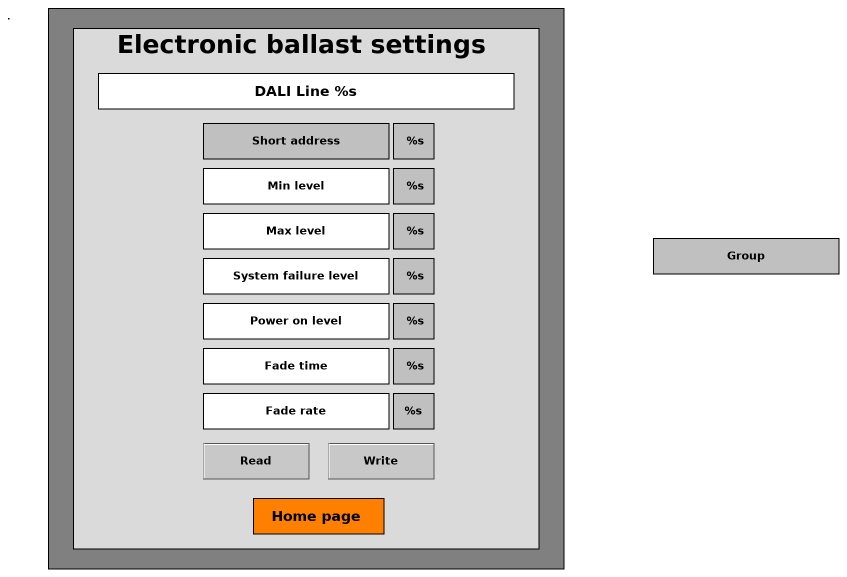
rectangle at (150,40)-(616,561): text "Electronic ballast settings"
rectangle at (280,225)-(466,261): text "Max level"
rectangle at (280,180)-(466,216): text "Min level"
rectangle at (280,270)-(466,306): text "System failure level"
rectangle at (280,315)-(466,351): text "Power on level"
rectangle at (280,360)-(466,396): text "Fade time"
rectangle at (280,405)-(466,441): text "Fade rate"
rectangle at (280,135)-(466,171): text "Short address"; invisible if DALI_Config.Kurzadr_Gruppe; toggles DALI_Config.Kurzadr_Gruppe
rectangle at (730,250)-(916,286): text "Group"; invisible if not DALI_Config.Kurzadr_Gruppe; toggles DALI_Config.Kurzadr_Gruppe; tooltip Selection group or short address
rectangle at (470,135)-(511,171): text "%s"; shows DALI_Config.Adresse; tooltip Enter group (1-16) or short address (1 - 64); editable
rounded rectangle at (330,510)-(461,546): text "Home page"; opens PLC_VISU; tooltip Back to home page
rectangle at (470,180)-(511,216): text "%s"; shows DALI_Config.MinLevel; tooltip Minimal brightness level in percent. Min level has to be smaller than max level.; editable
rectangle at (470,225)-(511,261): text "%s"; shows DALI_Config.MaxLevel; tooltip Maximum brightness level in percent; editable
rectangle at (470,270)-(511,306): text "%s"; shows DALI_Config.SystemFailure; tooltip Brightness level in percent in case of a system failure. The value 101 means "MASK".; editable
rectangle at (470,315)-(511,351): text "%s"; shows DALI_Config.PowerOn; tooltip Brightness level in percent if the ECGs are powered on.; editable
rectangle at (470,360)-(511,396): text "%s"; shows DALI_Config.Konfig[4]; tooltip Enter the fade time (0 - 15); editable
rectangle at (470,405)-(511,441): text "%s"; shows DALI_Config.Konfig[5]; tooltip Enter the fade rate (1 -15); editable
button at (280,455)-(386,491): text "Read"; taps DALI_Config.Lese; tooltip If you click the button "Read", the settings of the ECG will be read. Group queries are not possible.
button at (405,455)-(511,491): text "Write"; taps DALI_Config.Schreib; tooltip If you click the button "Write", the new settings will be written into the ECG.
rounded rectangle at (175,85)-(591,121): text "DALI Line %s"; shows DALI_Config.bDali_Linie; tooltip You can change the DALI Line only on the home page.
2 more shapes without text or variables
*)

(* Visualisation Group_assignment
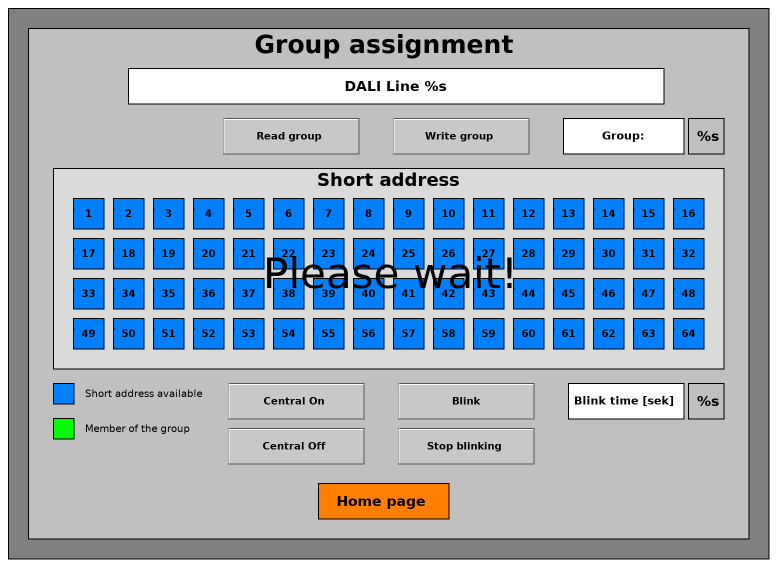
rectangle at (40,40)-(761,551): text "Group assignment"
rounded rectangle at (330,495)-(461,531): text "Home page"; opens PLC_VISU; tooltip Back to home page
rectangle at (65,180)-(736,381): text "Short address"
rectangle at (85,210)-(116,241): text "1"; alarm colour if DALI_Config.Kurzadr[1]
rectangle at (85,210)-(116,241): text "1"; invisible if not DALI_Config.Kurzadr[1]; alarm colour if DALI_Config.Gruppenadr[1]; toggles DALI_Config.Gruppenadr[1]
rectangle at (125,210)-(156,241): text "2"; alarm colour if DALI_Config.Kurzadr[2]
rectangle at (125,210)-(156,241): text "2"; invisible if not DALI_Config.Kurzadr[2]; alarm colour if DALI_Config.Gruppenadr[2]; toggles DALI_Config.Gruppenadr[2]
rectangle at (165,210)-(196,241): text "3"; alarm colour if DALI_Config.Kurzadr[3]
rectangle at (165,210)-(196,241): text "3"; invisible if not DALI_Config.Kurzadr[3]; alarm colour if DALI_Config.Gruppenadr[3]; toggles DALI_Config.Gruppenadr[3]
rectangle at (205,210)-(236,241): text "4"; alarm colour if DALI_Config.Kurzadr[4]
rectangle at (205,210)-(236,241): text "4"; invisible if not DALI_Config.Kurzadr[4]; alarm colour if DALI_Config.Gruppenadr[4]; toggles DALI_Config.Gruppenadr[4]
rectangle at (245,210)-(276,241): text "5"; alarm colour if DALI_Config.Kurzadr[5]
rectangle at (245,210)-(276,241): text "5"; invisible if not DALI_Config.Kurzadr[5]; alarm colour if DALI_Config.Gruppenadr[5]; toggles DALI_Config.Gruppenadr[5]
rectangle at (285,210)-(316,241): text "6"; alarm colour if DALI_Config.Kurzadr[6]
rectangle at (285,210)-(316,241): text "6"; invisible if not DALI_Config.Kurzadr[6]; alarm colour if DALI_Config.Gruppenadr[6]; toggles DALI_Config.Gruppenadr[6]
rectangle at (325,210)-(356,241): text "7"; alarm colour if DALI_Config.Kurzadr[7]
rectangle at (325,210)-(356,241): text "7"; invisible if not DALI_Config.Kurzadr[7]; alarm colour if DALI_Config.Gruppenadr[7]; toggles DALI_Config.Gruppenadr[7]
rectangle at (365,210)-(396,241): text "8"; alarm colour if DALI_Config.Kurzadr[8]
rectangle at (365,210)-(396,241): text "8"; invisible if not DALI_Config.Kurzadr[8]; alarm colour if DALI_Config.Gruppenadr[8]; toggles DALI_Config.Gruppenadr[8]
rectangle at (405,210)-(436,241): text "9"; alarm colour if DALI_Config.Kurzadr[9]
rectangle at (405,210)-(436,241): text "9"; invisible if not DALI_Config.Kurzadr[9]; alarm colour if DALI_Config.Gruppenadr[9]; toggles DALI_Config.Gruppenadr[9]
rectangle at (445,210)-(476,241): text "10"; alarm colour if DALI_Config.Kurzadr[10]
rectangle at (445,210)-(476,241): text "10"; invisible if not DALI_Config.Kurzadr[10]; alarm colour if DALI_Config.Gruppenadr[10]; toggles DALI_Config.Gruppenadr[10]
rectangle at (485,210)-(516,241): text "11"; alarm colour if DALI_Config.Kurzadr[11]
rectangle at (485,210)-(516,241): text "11"; invisible if not DALI_Config.Kurzadr[11]; alarm colour if DALI_Config.Gruppenadr[11]; toggles DALI_Config.Gruppenadr[11]
rectangle at (525,210)-(556,241): text "12"; alarm colour if DALI_Config.Kurzadr[12]
rectangle at (525,210)-(556,241): text "12"; invisible if not DALI_Config.Kurzadr[12]; alarm colour if DALI_Config.Gruppenadr[12]; toggles DALI_Config.Gruppenadr[12]
rectangle at (565,210)-(596,241): text "13"; alarm colour if DALI_Config.Kurzadr[13]
rectangle at (565,210)-(596,241): text "13"; invisible if not DALI_Config.Kurzadr[13]; alarm colour if DALI_Config.Gruppenadr[13]; toggles DALI_Config.Gruppenadr[13]
rectangle at (605,210)-(636,241): text "14"; alarm colour if DALI_Config.Kurzadr[14]
rectangle at (605,210)-(636,241): text "14"; invisible if not DALI_Config.Kurzadr[14]; alarm colour if DALI_Config.Gruppenadr[14]; toggles DALI_Config.Gruppenadr[14]
rectangle at (645,210)-(676,241): text "15"; alarm colour if DALI_Config.Kurzadr[15]
rectangle at (645,210)-(676,241): text "15"; invisible if not DALI_Config.Kurzadr[15]; alarm colour if DALI_Config.Gruppenadr[15]; toggles DALI_Config.Gruppenadr[15]
rectangle at (685,210)-(716,241): text "16"; alarm colour if DALI_Config.Kurzadr[16]
rectangle at (685,210)-(716,241): text "16"; invisible if not DALI_Config.Kurzadr[16]; alarm colour if DALI_Config.Gruppenadr[16]; toggles DALI_Config.Gruppenadr[16]
button at (405,130)-(541,166): text "Write group"; taps DALI_Config.Gruppenkonfiguration; tooltip If you click the button "Write Group", the marked short addresses will be saved as a group.
rectangle at (575,130)-(696,166): text "Group:"
rectangle at (700,130)-(736,166): text "%s"; shows DALI_Config.Gruppe; tooltip Enter the number of the group (1 - 16); editable
button at (410,395)-(546,431): text "Blink"; taps DALI_Config.BlinkenGruppe; tooltip If you click the button "Blink", the selected ECG will blink as long as defined by the "Blink Time" parameter.
button at (410,440)-(546,476): text "Stop blinking"; taps DALI_Config.xBlinken_Aus; tooltip If you click the button "Stop blinking", the blinking of the ECG will stop immediately.
button at (235,130)-(371,166): text "Read group"; taps DALI_Config.GruppeLesen; tooltip If you click the button "Read Group", the short addresses that belong to the group will be displayed.
rectangle at (95,395)-(226,416): text "Short address available"
rectangle at (95,430)-(246,451): text "Member of the group"
rounded rectangle at (140,80)-(676,116): text "DALI Line %s"; shows DALI_Config.bDali_Linie; tooltip You can change the DALI Line only on the home page.
rectangle at (85,250)-(116,281): text "17"; alarm colour if DALI_Config.Kurzadr[17]
rectangle at (85,250)-(116,281): text "17"; invisible if not DALI_Config.Kurzadr[17]; alarm colour if DALI_Config.Gruppenadr[17]; toggles DALI_Config.Gruppenadr[17]
rectangle at (125,250)-(156,281): text "18"; alarm colour if DALI_Config.Kurzadr[18]
rectangle at (125,250)-(156,281): text "18"; invisible if not DALI_Config.Kurzadr[18]; alarm colour if DALI_Config.Gruppenadr[18]; toggles DALI_Config.Gruppenadr[18]
rectangle at (165,250)-(196,281): text "19"; alarm colour if DALI_Config.Kurzadr[19]
rectangle at (165,250)-(196,281): text "19"; invisible if not DALI_Config.Kurzadr[19]; alarm colour if DALI_Config.Gruppenadr[19]; toggles DALI_Config.Gruppenadr[19]
rectangle at (205,250)-(236,281): text "20"; alarm colour if DALI_Config.Kurzadr[20]
rectangle at (205,250)-(236,281): text "20"; invisible if not DALI_Config.Kurzadr[20]; alarm colour if DALI_Config.Gruppenadr[20]; toggles DALI_Config.Gruppenadr[20]
rectangle at (245,250)-(276,281): text "21"; alarm colour if DALI_Config.Kurzadr[21]
rectangle at (245,250)-(276,281): text "21"; invisible if not DALI_Config.Kurzadr[21]; alarm colour if DALI_Config.Gruppenadr[21]; toggles DALI_Config.Gruppenadr[21]
rectangle at (285,250)-(316,281): text "22"; alarm colour if DALI_Config.Kurzadr[22]
rectangle at (285,250)-(316,281): text "22"; invisible if not DALI_Config.Kurzadr[22]; alarm colour if DALI_Config.Gruppenadr[22]; toggles DALI_Config.Gruppenadr[22]
rectangle at (325,250)-(356,281): text "23"; alarm colour if DALI_Config.Kurzadr[23]
rectangle at (325,250)-(356,281): text "23"; invisible if not DALI_Config.Kurzadr[23]; alarm colour if DALI_Config.Gruppenadr[23]; toggles DALI_Config.Gruppenadr[23]
rectangle at (365,250)-(396,281): text "24"; alarm colour if DALI_Config.Kurzadr[24]
rectangle at (365,250)-(396,281): text "24"; invisible if not DALI_Config.Kurzadr[24]; alarm colour if DALI_Config.Gruppenadr[24]; toggles DALI_Config.Gruppenadr[24]
rectangle at (405,250)-(436,281): text "25"; alarm colour if DALI_Config.Kurzadr[25]
rectangle at (405,250)-(436,281): text "25"; invisible if not DALI_Config.Kurzadr[25]; alarm colour if DALI_Config.Gruppenadr[25]; toggles DALI_Config.Gruppenadr[25]
rectangle at (445,250)-(476,281): text "26"; alarm colour if DALI_Config.Kurzadr[26]
rectangle at (445,250)-(476,281): text "26"; invisible if not DALI_Config.Kurzadr[26]; alarm colour if DALI_Config.Gruppenadr[26]; toggles DALI_Config.Gruppenadr[26]
rectangle at (485,250)-(516,281): text "27"; alarm colour if DALI_Config.Kurzadr[27]
rectangle at (485,250)-(516,281): text "27"; invisible if not DALI_Config.Kurzadr[27]; alarm colour if DALI_Config.Gruppenadr[27]; toggles DALI_Config.Gruppenadr[27]
rectangle at (525,250)-(556,281): text "28"; alarm colour if DALI_Config.Kurzadr[28]
rectangle at (525,250)-(556,281): text "28"; invisible if not DALI_Config.Kurzadr[28]; alarm colour if DALI_Config.Gruppenadr[28]; toggles DALI_Config.Gruppenadr[28]
rectangle at (565,250)-(596,281): text "29"; alarm colour if DALI_Config.Kurzadr[29]
rectangle at (565,250)-(596,281): text "29"; invisible if not DALI_Config.Kurzadr[29]; alarm colour if DALI_Config.Gruppenadr[29]; toggles DALI_Config.Gruppenadr[29]
rectangle at (605,250)-(636,281): text "30"; alarm colour if DALI_Config.Kurzadr[30]
rectangle at (605,250)-(636,281): text "30"; invisible if not DALI_Config.Kurzadr[30]; alarm colour if DALI_Config.Gruppenadr[30]; toggles DALI_Config.Gruppenadr[30]
rectangle at (645,250)-(676,281): text "31"; alarm colour if DALI_Config.Kurzadr[31]
rectangle at (645,250)-(676,281): text "31"; invisible if not DALI_Config.Kurzadr[31]; alarm colour if DALI_Config.Gruppenadr[31]; toggles DALI_Config.Gruppenadr[31]
rectangle at (685,250)-(716,281): text "32"; alarm colour if DALI_Config.Kurzadr[32]
rectangle at (685,250)-(716,281): text "32"; invisible if not DALI_Config.Kurzadr[32]; alarm colour if DALI_Config.Gruppenadr[32]; toggles DALI_Config.Gruppenadr[32]
rectangle at (85,290)-(116,321): text "33"; alarm colour if DALI_Config.Kurzadr[33]
rectangle at (85,290)-(116,321): text "33"; invisible if not DALI_Config.Kurzadr[33]; alarm colour if DALI_Config.Gruppenadr[33]; toggles DALI_Config.Gruppenadr[33]
rectangle at (125,290)-(156,321): text "34"; alarm colour if DALI_Config.Kurzadr[34]
rectangle at (125,290)-(156,321): text "34"; invisible if not DALI_Config.Kurzadr[34]; alarm colour if DALI_Config.Gruppenadr[34]; toggles DALI_Config.Gruppenadr[34]
rectangle at (165,290)-(196,321): text "35"; alarm colour if DALI_Config.Kurzadr[35]
rectangle at (165,290)-(196,321): text "35"; invisible if not DALI_Config.Kurzadr[35]; alarm colour if DALI_Config.Gruppenadr[35]; toggles DALI_Config.Gruppenadr[35]
rectangle at (205,290)-(236,321): text "36"; alarm colour if DALI_Config.Kurzadr[36]
rectangle at (205,290)-(236,321): text "36"; invisible if not DALI_Config.Kurzadr[36]; alarm colour if DALI_Config.Gruppenadr[36]; toggles DALI_Config.Gruppenadr[36]
rectangle at (245,290)-(276,321): text "37"; alarm colour if DALI_Config.Kurzadr[37]
rectangle at (245,290)-(276,321): text "37"; invisible if not DALI_Config.Kurzadr[37]; alarm colour if DALI_Config.Gruppenadr[37]; toggles DALI_Config.Gruppenadr[37]
rectangle at (285,290)-(316,321): text "38"; alarm colour if DALI_Config.Kurzadr[38]
rectangle at (285,290)-(316,321): text "38"; invisible if not DALI_Config.Kurzadr[38]; alarm colour if DALI_Config.Gruppenadr[38]; toggles DALI_Config.Gruppenadr[38]
rectangle at (325,290)-(356,321): text "39"; alarm colour if DALI_Config.Kurzadr[39]
rectangle at (325,290)-(356,321): text "39"; invisible if not DALI_Config.Kurzadr[39]; alarm colour if DALI_Config.Gruppenadr[39]; toggles DALI_Config.Gruppenadr[39]
rectangle at (365,290)-(396,321): text "40"; alarm colour if DALI_Config.Kurzadr[40]
rectangle at (365,290)-(396,321): text "40"; invisible if not DALI_Config.Kurzadr[40]; alarm colour if DALI_Config.Gruppenadr[40]; toggles DALI_Config.Gruppenadr[40]
rectangle at (405,290)-(436,321): text "41"; alarm colour if DALI_Config.Kurzadr[41]
rectangle at (405,290)-(436,321): text "41"; invisible if not DALI_Config.Kurzadr[41]; alarm colour if DALI_Config.Gruppenadr[41]; toggles DALI_Config.Gruppenadr[41]
rectangle at (445,290)-(476,321): text "42"; alarm colour if DALI_Config.Kurzadr[42]
rectangle at (445,290)-(476,321): text "42"; invisible if not DALI_Config.Kurzadr[42]; alarm colour if DALI_Config.Gruppenadr[42]; toggles DALI_Config.Gruppenadr[42]
rectangle at (485,290)-(516,321): text "43"; alarm colour if DALI_Config.Kurzadr[43]
rectangle at (485,290)-(516,321): text "43"; invisible if not DALI_Config.Kurzadr[43]; alarm colour if DALI_Config.Gruppenadr[43]; toggles DALI_Config.Gruppenadr[43]
rectangle at (525,290)-(556,321): text "44"; alarm colour if DALI_Config.Kurzadr[44]
rectangle at (525,290)-(556,321): text "44"; invisible if not DALI_Config.Kurzadr[44]; alarm colour if DALI_Config.Gruppenadr[44]; toggles DALI_Config.Gruppenadr[44]
rectangle at (565,290)-(596,321): text "45"; alarm colour if DALI_Config.Kurzadr[45]
rectangle at (565,290)-(596,321): text "45"; invisible if not DALI_Config.Kurzadr[45]; alarm colour if DALI_Config.Gruppenadr[45]; toggles DALI_Config.Gruppenadr[45]
rectangle at (605,290)-(636,321): text "46"; alarm colour if DALI_Config.Kurzadr[46]
rectangle at (605,290)-(636,321): text "46"; invisible if not DALI_Config.Kurzadr[46]; alarm colour if DALI_Config.Gruppenadr[46]; toggles DALI_Config.Gruppenadr[46]
rectangle at (645,290)-(676,321): text "47"; alarm colour if DALI_Config.Kurzadr[47]
rectangle at (645,290)-(676,321): text "47"; invisible if not DALI_Config.Kurzadr[47]; alarm colour if DALI_Config.Gruppenadr[47]; toggles DALI_Config.Gruppenadr[47]
rectangle at (685,290)-(716,321): text "48"; alarm colour if DALI_Config.Kurzadr[48]
rectangle at (685,290)-(716,321): text "48"; invisible if not DALI_Config.Kurzadr[48]; alarm colour if DALI_Config.Gruppenadr[48]; toggles DALI_Config.Gruppenadr[48]
rectangle at (85,330)-(116,361): text "49"; alarm colour if DALI_Config.Kurzadr[49]
rectangle at (85,330)-(116,361): text "49"; invisible if not DALI_Config.Kurzadr[49]; alarm colour if DALI_Config.Gruppenadr[49]; toggles DALI_Config.Gruppenadr[49]
rectangle at (125,330)-(156,361): text "50"; alarm colour if DALI_Config.Kurzadr[50]
rectangle at (125,330)-(156,361): text "50"; invisible if not DALI_Config.Kurzadr[50]; alarm colour if DALI_Config.Gruppenadr[50]; toggles DALI_Config.Gruppenadr[50]
rectangle at (165,330)-(196,361): text "51"; alarm colour if DALI_Config.Kurzadr[51]
rectangle at (165,330)-(196,361): text "51"; invisible if not DALI_Config.Kurzadr[51]; alarm colour if DALI_Config.Gruppenadr[51]; toggles DALI_Config.Gruppenadr[51]
rectangle at (205,330)-(236,361): text "52"; alarm colour if DALI_Config.Kurzadr[52]
rectangle at (205,330)-(236,361): text "52"; invisible if not DALI_Config.Kurzadr[52]; alarm colour if DALI_Config.Gruppenadr[52]; toggles DALI_Config.Gruppenadr[52]
rectangle at (245,330)-(276,361): text "53"; alarm colour if DALI_Config.Kurzadr[53]
rectangle at (245,330)-(276,361): text "53"; invisible if not DALI_Config.Kurzadr[53]; alarm colour if DALI_Config.Gruppenadr[53]; toggles DALI_Config.Gruppenadr[53]
rectangle at (285,330)-(316,361): text "54"; alarm colour if DALI_Config.Kurzadr[54]
rectangle at (285,330)-(316,361): text "54"; invisible if not DALI_Config.Kurzadr[54]; alarm colour if DALI_Config.Gruppenadr[54]; toggles DALI_Config.Gruppenadr[54]
rectangle at (325,330)-(356,361): text "55"; alarm colour if DALI_Config.Kurzadr[55]
rectangle at (325,330)-(356,361): text "55"; invisible if not DALI_Config.Kurzadr[55]; alarm colour if DALI_Config.Gruppenadr[55]; toggles DALI_Config.Gruppenadr[55]
rectangle at (365,330)-(396,361): text "56"; alarm colour if DALI_Config.Kurzadr[56]
rectangle at (365,330)-(396,361): text "56"; invisible if not DALI_Config.Kurzadr[56]; alarm colour if DALI_Config.Gruppenadr[56]; toggles DALI_Config.Gruppenadr[56]
rectangle at (405,330)-(436,361): text "57"; alarm colour if DALI_Config.Kurzadr[57]
rectangle at (405,330)-(436,361): text "57"; invisible if not DALI_Config.Kurzadr[57]; alarm colour if DALI_Config.Gruppenadr[57]; toggles DALI_Config.Gruppenadr[57]
rectangle at (445,330)-(476,361): text "58"; alarm colour if DALI_Config.Kurzadr[58]
rectangle at (445,330)-(476,361): text "58"; invisible if not DALI_Config.Kurzadr[58]; alarm colour if DALI_Config.Gruppenadr[58]; toggles DALI_Config.Gruppenadr[58]
rectangle at (485,330)-(516,361): text "59"; alarm colour if DALI_Config.Kurzadr[59]
rectangle at (485,330)-(516,361): text "59"; invisible if not DALI_Config.Kurzadr[59]; alarm colour if DALI_Config.Gruppenadr[59]; toggles DALI_Config.Gruppenadr[59]
rectangle at (525,330)-(556,361): text "60"; alarm colour if DALI_Config.Kurzadr[60]
rectangle at (525,330)-(556,361): text "60"; invisible if not DALI_Config.Kurzadr[60]; alarm colour if DALI_Config.Gruppenadr[60]; toggles DALI_Config.Gruppenadr[60]
rectangle at (565,330)-(596,361): text "61"; alarm colour if DALI_Config.Kurzadr[61]
rectangle at (565,330)-(596,361): text "61"; invisible if not DALI_Config.Kurzadr[61]; alarm colour if DALI_Config.Gruppenadr[61]; toggles DALI_Config.Gruppenadr[61]
rectangle at (605,330)-(636,361): text "62"; alarm colour if DALI_Config.Kurzadr[62]
rectangle at (605,330)-(636,361): text "62"; invisible if not DALI_Config.Kurzadr[62]; alarm colour if DALI_Config.Gruppenadr[62]; toggles DALI_Config.Gruppenadr[62]
rectangle at (645,330)-(676,361): text "63"; alarm colour if DALI_Config.Kurzadr[63]
rectangle at (645,330)-(676,361): text "63"; invisible if not DALI_Config.Kurzadr[63]; alarm colour if DALI_Config.Gruppenadr[63]; toggles DALI_Config.Gruppenadr[63]
rectangle at (685,330)-(716,361): text "64"; alarm colour if DALI_Config.Kurzadr[64]
rectangle at (685,330)-(716,361): text "64"; invisible if not DALI_Config.Kurzadr[64]; alarm colour if DALI_Config.Gruppenadr[64]; toggles DALI_Config.Gruppenadr[64]
rectangle at (580,395)-(696,431): text "Blink time [sek]"
button at (240,440)-(376,476): text "Central Off"; taps DALI_Config.Aus; tooltip If you click the button "Central Off", all lamps in the network will be switched off.
button at (240,395)-(376,431): text "Central On"; taps DALI_Config.Ein; tooltip If you click the button "Central On", all lamps in the network will be switched on.
rectangle at (700,395)-(736,431): text "%s"; shows DALI_Config.bBlinkzeit; tooltip Enter blink time (3 - 255 seconds); editable
rectangle at (42,88)-(763,482): text "Please wait!"; invisible if NOT DALI_Config.Unsichtbar
67 more shapes without text or variables
*)

(* Visualisation GroupSceneConfiguration
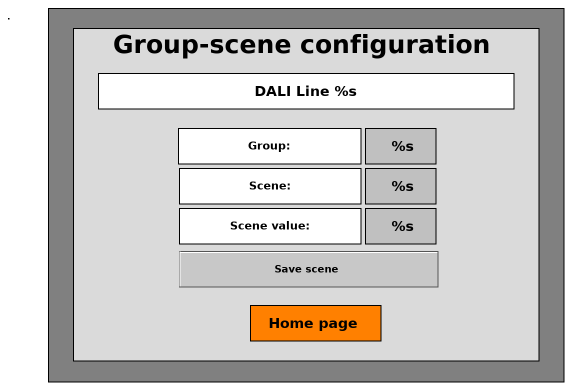
rectangle at (150,40)-(616,373): text "Group-scene configuration"
rounded rectangle at (327,317)-(458,353): text "Home page"; opens PLC_VISU; tooltip Back to home page
rounded rectangle at (175,85)-(591,121): text "DALI Line %s"; shows DALI_Config.bDali_Linie; tooltip You can change the DALI Line only on the home page.
rectangle at (255,140)-(438,176): text "Group:"
rectangle at (442,140)-(513,176): text "%s"; shows DALI_Config.sGroup; tooltip Enter the number of the group (1 - 16); editable
button at (256,263)-(515,299): text "Save scene"; taps DALI_Config.sSaveScene; tooltip Save the configured dim levels in the ECGs.
rectangle at (256,180)-(438,216): text "Scene:"
rectangle at (442,180)-(513,216): text "%s"; shows DALI_Config.sScene; tooltip Select scene 1 - 16; editable
rectangle at (256,220)-(438,256): text "Scene value:"
rectangle at (442,220)-(513,256): text "%s"; shows DALI_Config.sSceneValue; tooltip Select scene 1 - 16; editable
2 more shapes without text or variables
*)

(* Visualisation Lamp_status
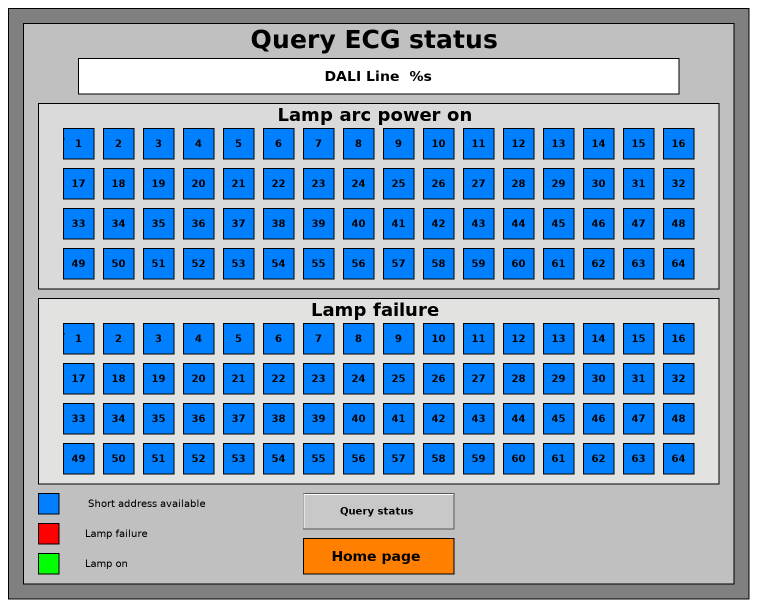
rectangle at (45,15)-(756,576): text "Query ECG status"
rounded rectangle at (325,530)-(476,566): text "Home page"; opens PLC_VISU; tooltip Back to home page
rounded rectangle at (100,50)-(701,86): text "DALI Line  %s"; shows DALI_Config.bDali_Linie; tooltip You can change the DALI Line only on the home page.
rectangle at (60,95)-(741,281): text "Lamp arc power on"
rectangle at (85,120)-(116,151): text "1"; alarm colour if DALI_Config.Kurzadr[1]
rectangle at (85,120)-(116,151): text "1"; invisible if not DALI_Config.Kurzadr[1]; alarm colour if DALI_Config.LampeEin[1]
rectangle at (125,120)-(156,151): text "2"; alarm colour if DALI_Config.Kurzadr[2]
rectangle at (125,120)-(156,151): text "2"; invisible if not DALI_Config.Kurzadr[2]; alarm colour if DALI_Config.LampeEin[2]
rectangle at (165,120)-(196,151): text "3"; alarm colour if DALI_Config.Kurzadr[3]
rectangle at (165,120)-(196,151): text "3"; invisible if not DALI_Config.Kurzadr[3]; alarm colour if DALI_Config.LampeEin[3]
rectangle at (205,120)-(236,151): text "4"; alarm colour if DALI_Config.Kurzadr[4]
rectangle at (205,120)-(236,151): text "4"; invisible if not DALI_Config.Kurzadr[4]; alarm colour if DALI_Config.LampeEin[4]
rectangle at (245,120)-(276,151): text "5"; alarm colour if DALI_Config.Kurzadr[5]
rectangle at (245,120)-(276,151): text "5"; invisible if not DALI_Config.Kurzadr[5]; alarm colour if DALI_Config.LampeEin[5]
rectangle at (285,120)-(316,151): text "6"; alarm colour if DALI_Config.Kurzadr[6]
rectangle at (285,120)-(316,151): text "6"; invisible if not DALI_Config.Kurzadr[6]; alarm colour if DALI_Config.LampeEin[6]
rectangle at (325,120)-(356,151): text "7"; alarm colour if DALI_Config.Kurzadr[7]
rectangle at (325,120)-(356,151): text "7"; invisible if not DALI_Config.Kurzadr[7]; alarm colour if DALI_Config.LampeEin[7]
rectangle at (365,120)-(396,151): text "8"; alarm colour if DALI_Config.Kurzadr[8]
rectangle at (365,120)-(396,151): text "8"; invisible if not DALI_Config.Kurzadr[8]; alarm colour if DALI_Config.LampeEin[8]
rectangle at (405,120)-(436,151): text "9"; alarm colour if DALI_Config.Kurzadr[9]
rectangle at (405,120)-(436,151): text "9"; invisible if not DALI_Config.Kurzadr[9]; alarm colour if DALI_Config.LampeEin[9]
rectangle at (445,120)-(476,151): text "10"; alarm colour if DALI_Config.Kurzadr[10]
rectangle at (445,120)-(476,151): text "10"; invisible if not DALI_Config.Kurzadr[10]; alarm colour if DALI_Config.LampeEin[10]
rectangle at (485,120)-(516,151): text "11"; alarm colour if DALI_Config.Kurzadr[11]
rectangle at (485,120)-(516,151): text "11"; invisible if not DALI_Config.Kurzadr[11]; alarm colour if DALI_Config.LampeEin[11]
rectangle at (525,120)-(556,151): text "12"; alarm colour if DALI_Config.Kurzadr[12]
rectangle at (525,120)-(556,151): text "12"; invisible if not DALI_Config.Kurzadr[12]; alarm colour if DALI_Config.LampeEin[12]
rectangle at (565,120)-(596,151): text "13"; alarm colour if DALI_Config.Kurzadr[13]
rectangle at (565,120)-(596,151): text "13"; invisible if not DALI_Config.Kurzadr[13]; alarm colour if DALI_Config.LampeEin[13]
rectangle at (605,120)-(636,151): text "14"; alarm colour if DALI_Config.Kurzadr[14]
rectangle at (605,120)-(636,151): text "14"; invisible if not DALI_Config.Kurzadr[14]; alarm colour if DALI_Config.LampeEin[14]
rectangle at (645,120)-(676,151): text "15"; alarm colour if DALI_Config.Kurzadr[15]
rectangle at (645,120)-(676,151): text "15"; invisible if not DALI_Config.Kurzadr[15]; alarm colour if DALI_Config.LampeEin[15]
rectangle at (685,120)-(716,151): text "16"; alarm colour if DALI_Config.Kurzadr[16]
rectangle at (685,120)-(716,151): text "16"; invisible if not DALI_Config.Kurzadr[16]; alarm colour if DALI_Config.LampeEin[16]
rectangle at (85,160)-(116,191): text "17"; alarm colour if DALI_Config.Kurzadr[17]
rectangle at (85,160)-(116,191): text "17"; invisible if not DALI_Config.Kurzadr[17]; alarm colour if DALI_Config.LampeEin[17]
rectangle at (165,160)-(196,191): text "19"; alarm colour if DALI_Config.Kurzadr[19]
rectangle at (165,160)-(196,191): text "19"; invisible if not DALI_Config.Kurzadr[19]; alarm colour if DALI_Config.LampeEin[19]
rectangle at (125,160)-(156,191): text "18"; alarm colour if DALI_Config.Kurzadr[18]
rectangle at (125,160)-(156,191): text "18"; invisible if not DALI_Config.Kurzadr[18]; alarm colour if DALI_Config.LampeEin[18]
rectangle at (205,160)-(236,191): text "20"; alarm colour if DALI_Config.Kurzadr[20]
rectangle at (205,160)-(236,191): text "20"; invisible if not DALI_Config.Kurzadr[20]; alarm colour if DALI_Config.LampeEin[20]
rectangle at (245,160)-(276,191): text "21"; alarm colour if DALI_Config.Kurzadr[21]
rectangle at (245,160)-(276,191): text "21"; invisible if not DALI_Config.Kurzadr[21]; alarm colour if DALI_Config.LampeEin[21]
rectangle at (285,160)-(316,191): text "22"; alarm colour if DALI_Config.Kurzadr[22]
rectangle at (285,160)-(316,191): text "22"; invisible if not DALI_Config.Kurzadr[22]; alarm colour if DALI_Config.LampeEin[22]
rectangle at (325,160)-(356,191): text "23"; alarm colour if DALI_Config.Kurzadr[23]
rectangle at (325,160)-(356,191): text "23"; invisible if not DALI_Config.Kurzadr[23]; alarm colour if DALI_Config.LampeEin[23]
rectangle at (365,160)-(396,191): text "24"; alarm colour if DALI_Config.Kurzadr[24]
rectangle at (365,160)-(396,191): text "24"; invisible if not DALI_Config.Kurzadr[24]; alarm colour if DALI_Config.LampeEin[24]
rectangle at (405,160)-(436,191): text "25"; alarm colour if DALI_Config.Kurzadr[25]
rectangle at (405,160)-(436,191): text "25"; invisible if not DALI_Config.Kurzadr[25]; alarm colour if DALI_Config.LampeEin[25]
rectangle at (565,160)-(596,191): text "29"; alarm colour if DALI_Config.Kurzadr[29]
rectangle at (565,160)-(596,191): text "29"; invisible if not DALI_Config.Kurzadr[29]; alarm colour if DALI_Config.LampeEin[29]
rectangle at (525,160)-(556,191): text "28"; alarm colour if DALI_Config.Kurzadr[28]
rectangle at (525,160)-(556,191): text "28"; invisible if not DALI_Config.Kurzadr[28]; alarm colour if DALI_Config.LampeEin[28]
rectangle at (485,160)-(516,191): text "27"; alarm colour if DALI_Config.Kurzadr[27]
rectangle at (485,160)-(516,191): text "27"; invisible if not DALI_Config.Kurzadr[27]; alarm colour if DALI_Config.LampeEin[27]
rectangle at (445,160)-(476,191): text "26"; alarm colour if DALI_Config.Kurzadr[26]
rectangle at (445,160)-(476,191): text "26"; invisible if not DALI_Config.Kurzadr[26]; alarm colour if DALI_Config.LampeEin[26]
rectangle at (605,160)-(636,191): text "30"; alarm colour if DALI_Config.Kurzadr[30]
rectangle at (605,160)-(636,191): text "30"; invisible if not DALI_Config.Kurzadr[30]; alarm colour if DALI_Config.LampeEin[30]
rectangle at (645,160)-(676,191): text "31"; alarm colour if DALI_Config.Kurzadr[31]
rectangle at (645,160)-(676,191): text "31"; invisible if not DALI_Config.Kurzadr[31]; alarm colour if DALI_Config.LampeEin[31]
rectangle at (685,160)-(716,191): text "32"; alarm colour if DALI_Config.Kurzadr[32]
rectangle at (685,160)-(716,191): text "32"; invisible if not DALI_Config.Kurzadr[32]; alarm colour if DALI_Config.LampeEin[32]
rectangle at (85,200)-(116,231): text "33"; alarm colour if DALI_Config.Kurzadr[33]
rectangle at (85,200)-(116,231): text "33"; invisible if not DALI_Config.Kurzadr[33]; alarm colour if DALI_Config.LampeEin[33]
rectangle at (125,200)-(156,231): text "34"; alarm colour if DALI_Config.Kurzadr[34]
rectangle at (125,200)-(156,231): text "34"; invisible if not DALI_Config.Kurzadr[34]; alarm colour if DALI_Config.LampeEin[34]
rectangle at (205,200)-(236,231): text "36"; alarm colour if DALI_Config.Kurzadr[36]
rectangle at (205,200)-(236,231): text "36"; invisible if not DALI_Config.Kurzadr[36]; alarm colour if DALI_Config.LampeEin[36]
rectangle at (285,200)-(316,231): text "38"; alarm colour if DALI_Config.Kurzadr[38]
rectangle at (285,200)-(316,231): text "38"; invisible if not DALI_Config.Kurzadr[38]; alarm colour if DALI_Config.LampeEin[38]
rectangle at (325,200)-(356,231): text "39"; alarm colour if DALI_Config.Kurzadr[39]
rectangle at (325,200)-(356,231): text "39"; invisible if not DALI_Config.Kurzadr[39]; alarm colour if DALI_Config.LampeEin[39]
rectangle at (245,200)-(276,231): text "37"; alarm colour if DALI_Config.Kurzadr[37]
rectangle at (245,200)-(276,231): text "37"; invisible if not DALI_Config.Kurzadr[37]; alarm colour if DALI_Config.LampeEin[37]
rectangle at (165,200)-(196,231): text "35"; alarm colour if DALI_Config.Kurzadr[35]
rectangle at (165,200)-(196,231): text "35"; invisible if not DALI_Config.Kurzadr[35]; alarm colour if DALI_Config.LampeEin[35]
rectangle at (405,200)-(436,231): text "41"; alarm colour if DALI_Config.Kurzadr[41]
rectangle at (405,200)-(436,231): text "41"; invisible if not DALI_Config.Kurzadr[41]; alarm colour if DALI_Config.LampeEin[41]
rectangle at (445,200)-(476,231): text "42"; alarm colour if DALI_Config.Kurzadr[42]
rectangle at (445,200)-(476,231): text "42"; invisible if not DALI_Config.Kurzadr[42]; alarm colour if DALI_Config.LampeEin[42]
rectangle at (365,200)-(396,231): text "40"; alarm colour if DALI_Config.Kurzadr[40]
rectangle at (365,200)-(396,231): text "40"; invisible if not DALI_Config.Kurzadr[40]; alarm colour if DALI_Config.LampeEin[40]
rectangle at (485,200)-(516,231): text "43"; alarm colour if DALI_Config.Kurzadr[43]
rectangle at (485,200)-(516,231): text "43"; invisible if not DALI_Config.Kurzadr[43]; alarm colour if DALI_Config.LampeEin[43]
rectangle at (525,200)-(556,231): text "44"; alarm colour if DALI_Config.Kurzadr[44]
rectangle at (525,200)-(556,231): text "44"; invisible if not DALI_Config.Kurzadr[44]; alarm colour if DALI_Config.LampeEin[44]
rectangle at (565,200)-(596,231): text "45"; alarm colour if DALI_Config.Kurzadr[45]
rectangle at (565,200)-(596,231): text "45"; invisible if not DALI_Config.Kurzadr[45]; alarm colour if DALI_Config.LampeEin[45]
rectangle at (605,200)-(636,231): text "46"; alarm colour if DALI_Config.Kurzadr[46]
rectangle at (605,200)-(636,231): text "46"; invisible if not DALI_Config.Kurzadr[46]; alarm colour if DALI_Config.LampeEin[46]
rectangle at (645,200)-(676,231): text "47"; alarm colour if DALI_Config.Kurzadr[47]
rectangle at (645,200)-(676,231): text "47"; invisible if not DALI_Config.Kurzadr[47]; alarm colour if DALI_Config.LampeEin[47]
rectangle at (685,200)-(716,231): text "48"; alarm colour if DALI_Config.Kurzadr[48]
rectangle at (685,200)-(716,231): text "48"; invisible if not DALI_Config.Kurzadr[48]; alarm colour if DALI_Config.LampeEin[48]
rectangle at (85,240)-(116,271): text "49"; alarm colour if DALI_Config.Kurzadr[49]
rectangle at (85,240)-(116,271): text "49"; invisible if not DALI_Config.Kurzadr[49]; alarm colour if DALI_Config.LampeEin[49]
rectangle at (125,240)-(156,271): text "50"; alarm colour if DALI_Config.Kurzadr[50]
rectangle at (125,240)-(156,271): text "50"; invisible if not DALI_Config.Kurzadr[50]; alarm colour if DALI_Config.LampeEin[50]
rectangle at (165,240)-(196,271): text "51"; alarm colour if DALI_Config.Kurzadr[51]
rectangle at (165,240)-(196,271): text "51"; invisible if not DALI_Config.Kurzadr[51]; alarm colour if DALI_Config.LampeEin[51]
rectangle at (205,240)-(236,271): text "52"; alarm colour if DALI_Config.Kurzadr[52]
rectangle at (205,240)-(236,271): text "52"; invisible if not DALI_Config.Kurzadr[52]; alarm colour if DALI_Config.LampeEin[52]
rectangle at (245,240)-(276,271): text "53"; alarm colour if DALI_Config.Kurzadr[53]
rectangle at (245,240)-(276,271): text "53"; invisible if not DALI_Config.Kurzadr[53]; alarm colour if DALI_Config.LampeEin[53]
rectangle at (285,240)-(316,271): text "54"; alarm colour if DALI_Config.Kurzadr[54]
rectangle at (285,240)-(316,271): text "54"; invisible if not DALI_Config.Kurzadr[54]; alarm colour if DALI_Config.LampeEin[54]
rectangle at (325,240)-(356,271): text "55"; alarm colour if DALI_Config.Kurzadr[55]
rectangle at (325,240)-(356,271): text "55"; invisible if not DALI_Config.Kurzadr[55]; alarm colour if DALI_Config.LampeEin[55]
rectangle at (365,240)-(396,271): text "56"; alarm colour if DALI_Config.Kurzadr[56]
rectangle at (365,240)-(396,271): text "56"; invisible if not DALI_Config.Kurzadr[56]; alarm colour if DALI_Config.LampeEin[56]
rectangle at (405,240)-(436,271): text "57"; alarm colour if DALI_Config.Kurzadr[57]
rectangle at (405,240)-(436,271): text "57"; invisible if not DALI_Config.Kurzadr[57]; alarm colour if DALI_Config.LampeEin[57]
rectangle at (485,240)-(516,271): text "59"; alarm colour if DALI_Config.Kurzadr[59]
rectangle at (485,240)-(516,271): text "59"; invisible if not DALI_Config.Kurzadr[59]; alarm colour if DALI_Config.LampeEin[59]
rectangle at (525,240)-(556,271): text "60"; alarm colour if DALI_Config.Kurzadr[60]
rectangle at (525,240)-(556,271): text "60"; invisible if not DALI_Config.Kurzadr[60]; alarm colour if DALI_Config.LampeEin[60]
rectangle at (565,240)-(596,271): text "61"; alarm colour if DALI_Config.Kurzadr[61]
rectangle at (565,240)-(596,271): text "61"; invisible if not DALI_Config.Kurzadr[61]; alarm colour if DALI_Config.LampeEin[61]
rectangle at (605,240)-(636,271): text "62"; alarm colour if DALI_Config.Kurzadr[62]
rectangle at (605,240)-(636,271): text "62"; invisible if not DALI_Config.Kurzadr[62]; alarm colour if DALI_Config.LampeEin[62]
rectangle at (445,240)-(476,271): text "58"; alarm colour if DALI_Config.Kurzadr[58]
rectangle at (445,240)-(476,271): text "58"; invisible if not DALI_Config.Kurzadr[58]; alarm colour if DALI_Config.LampeEin[58]
rectangle at (645,240)-(676,271): text "63"; alarm colour if DALI_Config.Kurzadr[63]
rectangle at (645,240)-(676,271): text "63"; invisible if not DALI_Config.Kurzadr[63]; alarm colour if DALI_Config.LampeEin[63]
rectangle at (685,240)-(716,271): text "64"; alarm colour if DALI_Config.Kurzadr[64]
rectangle at (685,240)-(716,271): text "64"; invisible if not DALI_Config.Kurzadr[64]; alarm colour if DALI_Config.LampeEin[64]
rectangle at (60,290)-(741,476): text "Lamp failure"
rectangle at (85,315)-(116,346): text "1"; alarm colour if DALI_Config.Kurzadr[1]
rectangle at (85,315)-(116,346): text "1"; invisible if not DALI_Config.Kurzadr[1]; alarm colour if DALI_Config.Lampenausfall[1]
rectangle at (125,315)-(156,346): text "2"; alarm colour if DALI_Config.Kurzadr[2]
rectangle at (125,315)-(156,346): text "2"; invisible if not DALI_Config.Kurzadr[2]; alarm colour if DALI_Config.Lampenausfall[2]
rectangle at (165,315)-(196,346): text "3"; alarm colour if DALI_Config.Kurzadr[3]
rectangle at (165,315)-(196,346): text "3"; invisible if not DALI_Config.Kurzadr[3]; alarm colour if DALI_Config.Lampenausfall[3]
rectangle at (205,315)-(236,346): text "4"; alarm colour if DALI_Config.Kurzadr[4]
rectangle at (205,315)-(236,346): text "4"; invisible if not DALI_Config.Kurzadr[4]; alarm colour if DALI_Config.Lampenausfall[4]
rectangle at (245,315)-(276,346): text "5"; alarm colour if DALI_Config.Kurzadr[5]
rectangle at (245,315)-(276,346): text "5"; invisible if not DALI_Config.Kurzadr[5]; alarm colour if DALI_Config.Lampenausfall[5]
rectangle at (285,315)-(316,346): text "6"; alarm colour if DALI_Config.Kurzadr[6]
rectangle at (285,315)-(316,346): text "6"; invisible if not DALI_Config.Kurzadr[6]; alarm colour if DALI_Config.Lampenausfall[6]
rectangle at (325,315)-(356,346): text "7"; alarm colour if DALI_Config.Kurzadr[7]
rectangle at (325,315)-(356,346): text "7"; invisible if not DALI_Config.Kurzadr[7]; alarm colour if DALI_Config.Lampenausfall[7]
rectangle at (365,315)-(396,346): text "8"; alarm colour if DALI_Config.Kurzadr[8]
rectangle at (365,315)-(396,346): text "8"; invisible if not DALI_Config.Kurzadr[8]; alarm colour if DALI_Config.Lampenausfall[8]
rectangle at (405,315)-(436,346): text "9"; alarm colour if DALI_Config.Kurzadr[9]
rectangle at (405,315)-(436,346): text "9"; invisible if not DALI_Config.Kurzadr[9]; alarm colour if DALI_Config.Lampenausfall[9]
rectangle at (445,315)-(476,346): text "10"; alarm colour if DALI_Config.Kurzadr[10]
rectangle at (445,315)-(476,346): text "10"; invisible if not DALI_Config.Kurzadr[10]; alarm colour if DALI_Config.Lampenausfall[10]
rectangle at (485,315)-(516,346): text "11"; alarm colour if DALI_Config.Kurzadr[11]
rectangle at (485,315)-(516,346): text "11"; invisible if not DALI_Config.Kurzadr[11]; alarm colour if DALI_Config.Lampenausfall[11]
rectangle at (525,315)-(556,346): text "12"; alarm colour if DALI_Config.Kurzadr[12]
rectangle at (525,315)-(556,346): text "12"; invisible if not DALI_Config.Kurzadr[12]; alarm colour if DALI_Config.Lampenausfall[12]
rectangle at (565,315)-(596,346): text "13"; alarm colour if DALI_Config.Kurzadr[13]
rectangle at (565,315)-(596,346): text "13"; invisible if not DALI_Config.Kurzadr[13]; alarm colour if DALI_Config.Lampenausfall[13]
rectangle at (605,315)-(636,346): text "14"; alarm colour if DALI_Config.Kurzadr[14]
rectangle at (605,315)-(636,346): text "14"; invisible if not DALI_Config.Kurzadr[14]; alarm colour if DALI_Config.Lampenausfall[14]
rectangle at (645,315)-(676,346): text "15"; alarm colour if DALI_Config.Kurzadr[15]
rectangle at (645,315)-(676,346): text "15"; invisible if not DALI_Config.Kurzadr[15]; alarm colour if DALI_Config.Lampenausfall[15]
rectangle at (685,315)-(716,346): text "16"; alarm colour if DALI_Config.Kurzadr[16]
rectangle at (685,315)-(716,346): text "16"; invisible if not DALI_Config.Kurzadr[16]; alarm colour if DALI_Config.Lampenausfall[16]
rectangle at (85,355)-(116,386): text "17"; alarm colour if DALI_Config.Kurzadr[17]
rectangle at (85,355)-(116,386): text "17"; invisible if not DALI_Config.Kurzadr[17]; alarm colour if DALI_Config.Lampenausfall[17]
rectangle at (165,355)-(196,386): text "19"; alarm colour if DALI_Config.Kurzadr[19]
rectangle at (165,355)-(196,386): text "19"; invisible if not DALI_Config.Kurzadr[19]; alarm colour if DALI_Config.Lampenausfall[19]
rectangle at (125,355)-(156,386): text "18"; alarm colour if DALI_Config.Kurzadr[18]
rectangle at (125,355)-(156,386): text "18"; invisible if not DALI_Config.Kurzadr[18]; alarm colour if DALI_Config.Lampenausfall[18]
rectangle at (205,355)-(236,386): text "20"; alarm colour if DALI_Config.Kurzadr[20]
rectangle at (205,355)-(236,386): text "20"; invisible if not DALI_Config.Kurzadr[20]; alarm colour if DALI_Config.Lampenausfall[20]
rectangle at (245,355)-(276,386): text "21"; alarm colour if DALI_Config.Kurzadr[21]
rectangle at (245,355)-(276,386): text "21"; invisible if not DALI_Config.Kurzadr[21]; alarm colour if DALI_Config.Lampenausfall[21]
rectangle at (285,355)-(316,386): text "22"; alarm colour if DALI_Config.Kurzadr[22]
rectangle at (285,355)-(316,386): text "22"; invisible if not DALI_Config.Kurzadr[22]; alarm colour if DALI_Config.Lampenausfall[22]
rectangle at (325,355)-(356,386): text "23"; alarm colour if DALI_Config.Kurzadr[23]
rectangle at (325,355)-(356,386): text "23"; invisible if not DALI_Config.Kurzadr[23]; alarm colour if DALI_Config.Lampenausfall[23]
rectangle at (365,355)-(396,386): text "24"; alarm colour if DALI_Config.Kurzadr[24]
rectangle at (365,355)-(396,386): text "24"; invisible if not DALI_Config.Kurzadr[24]; alarm colour if DALI_Config.Lampenausfall[24]
rectangle at (405,355)-(436,386): text "25"; alarm colour if DALI_Config.Kurzadr[25]
rectangle at (405,355)-(436,386): text "25"; invisible if not DALI_Config.Kurzadr[25]; alarm colour if DALI_Config.Lampenausfall[25]
rectangle at (565,355)-(596,386): text "29"; alarm colour if DALI_Config.Kurzadr[29]
rectangle at (565,355)-(596,386): text "29"; invisible if not DALI_Config.Kurzadr[29]; alarm colour if DALI_Config.Lampenausfall[29]
rectangle at (525,355)-(556,386): text "28"; alarm colour if DALI_Config.Kurzadr[28]
rectangle at (525,355)-(556,386): text "28"; invisible if not DALI_Config.Kurzadr[28]; alarm colour if DALI_Config.Lampenausfall[28]
rectangle at (485,355)-(516,386): text "27"; alarm colour if DALI_Config.Kurzadr[27]
rectangle at (485,355)-(516,386): text "27"; invisible if not DALI_Config.Kurzadr[27]; alarm colour if DALI_Config.Lampenausfall[27]
rectangle at (445,355)-(476,386): text "26"; alarm colour if DALI_Config.Kurzadr[26]
rectangle at (445,355)-(476,386): text "26"; invisible if not DALI_Config.Kurzadr[26]; alarm colour if DALI_Config.Lampenausfall[26]
rectangle at (605,355)-(636,386): text "30"; alarm colour if DALI_Config.Kurzadr[30]
rectangle at (605,355)-(636,386): text "30"; invisible if not DALI_Config.Kurzadr[30]; alarm colour if DALI_Config.Lampenausfall[30]
rectangle at (645,355)-(676,386): text "31"; alarm colour if DALI_Config.Kurzadr[31]
rectangle at (645,355)-(676,386): text "31"; invisible if not DALI_Config.Kurzadr[31]; alarm colour if DALI_Config.Lampenausfall[31]
rectangle at (685,355)-(716,386): text "32"; alarm colour if DALI_Config.Kurzadr[32]
rectangle at (685,355)-(716,386): text "32"; invisible if not DALI_Config.Kurzadr[32]; alarm colour if DALI_Config.Lampenausfall[32]
rectangle at (85,395)-(116,426): text "33"; alarm colour if DALI_Config.Kurzadr[33]
rectangle at (85,395)-(116,426): text "33"; invisible if not DALI_Config.Kurzadr[33]; alarm colour if DALI_Config.Lampenausfall[33]
rectangle at (125,395)-(156,426): text "34"; alarm colour if DALI_Config.Kurzadr[34]
rectangle at (125,395)-(156,426): text "34"; invisible if not DALI_Config.Kurzadr[34]; alarm colour if DALI_Config.Lampenausfall[34]
rectangle at (205,395)-(236,426): text "36"; alarm colour if DALI_Config.Kurzadr[36]
rectangle at (205,395)-(236,426): text "36"; invisible if not DALI_Config.Kurzadr[36]; alarm colour if DALI_Config.Lampenausfall[36]
rectangle at (285,395)-(316,426): text "38"; alarm colour if DALI_Config.Kurzadr[38]
rectangle at (285,395)-(316,426): text "38"; invisible if not DALI_Config.Kurzadr[38]; alarm colour if DALI_Config.Lampenausfall[38]
rectangle at (325,395)-(356,426): text "39"; alarm colour if DALI_Config.Kurzadr[39]
rectangle at (325,395)-(356,426): text "39"; invisible if not DALI_Config.Kurzadr[39]; alarm colour if DALI_Config.Lampenausfall[39]
rectangle at (245,395)-(276,426): text "37"; alarm colour if DALI_Config.Kurzadr[37]
rectangle at (245,395)-(276,426): text "37"; invisible if not DALI_Config.Kurzadr[37]; alarm colour if DALI_Config.Lampenausfall[37]
rectangle at (165,395)-(196,426): text "35"; alarm colour if DALI_Config.Kurzadr[35]
rectangle at (165,395)-(196,426): text "35"; invisible if not DALI_Config.Kurzadr[35]; alarm colour if DALI_Config.Lampenausfall[35]
rectangle at (405,395)-(436,426): text "41"; alarm colour if DALI_Config.Kurzadr[41]
rectangle at (405,395)-(436,426): text "41"; invisible if not DALI_Config.Kurzadr[41]; alarm colour if DALI_Config.Lampenausfall[41]
rectangle at (445,395)-(476,426): text "42"; alarm colour if DALI_Config.Kurzadr[42]
rectangle at (445,395)-(476,426): text "42"; invisible if not DALI_Config.Kurzadr[42]; alarm colour if DALI_Config.Lampenausfall[42]
rectangle at (365,395)-(396,426): text "40"; alarm colour if DALI_Config.Kurzadr[40]
rectangle at (365,395)-(396,426): text "40"; invisible if not DALI_Config.Kurzadr[40]; alarm colour if DALI_Config.Lampenausfall[40]
rectangle at (485,395)-(516,426): text "43"; alarm colour if DALI_Config.Kurzadr[43]
rectangle at (485,395)-(516,426): text "43"; invisible if not DALI_Config.Kurzadr[43]; alarm colour if DALI_Config.Lampenausfall[43]
rectangle at (525,395)-(556,426): text "44"; alarm colour if DALI_Config.Kurzadr[44]
rectangle at (525,395)-(556,426): text "44"; invisible if not DALI_Config.Kurzadr[44]; alarm colour if DALI_Config.Lampenausfall[44]
rectangle at (565,395)-(596,426): text "45"; alarm colour if DALI_Config.Kurzadr[45]
rectangle at (565,395)-(596,426): text "45"; invisible if not DALI_Config.Kurzadr[45]; alarm colour if DALI_Config.Lampenausfall[45]
rectangle at (605,395)-(636,426): text "46"; alarm colour if DALI_Config.Kurzadr[46]
rectangle at (605,395)-(636,426): text "46"; invisible if not DALI_Config.Kurzadr[46]; alarm colour if DALI_Config.Lampenausfall[46]
rectangle at (645,395)-(676,426): text "47"; alarm colour if DALI_Config.Kurzadr[47]
rectangle at (645,395)-(676,426): text "47"; invisible if not DALI_Config.Kurzadr[47]; alarm colour if DALI_Config.Lampenausfall[47]
rectangle at (685,395)-(716,426): text "48"; alarm colour if DALI_Config.Kurzadr[48]
rectangle at (685,395)-(716,426): text "48"; invisible if not DALI_Config.Kurzadr[48]; alarm colour if DALI_Config.Lampenausfall[48]
rectangle at (85,435)-(116,466): text "49"; alarm colour if DALI_Config.Kurzadr[49]
rectangle at (85,435)-(116,466): text "49"; invisible if not DALI_Config.Kurzadr[49]; alarm colour if DALI_Config.Lampenausfall[49]
rectangle at (125,435)-(156,466): text "50"; alarm colour if DALI_Config.Kurzadr[50]
rectangle at (125,435)-(156,466): text "50"; invisible if not DALI_Config.Kurzadr[50]; alarm colour if DALI_Config.Lampenausfall[50]
rectangle at (165,435)-(196,466): text "51"; alarm colour if DALI_Config.Kurzadr[51]
rectangle at (165,435)-(196,466): text "51"; invisible if not DALI_Config.Kurzadr[51]; alarm colour if DALI_Config.Lampenausfall[51]
rectangle at (205,435)-(236,466): text "52"; alarm colour if DALI_Config.Kurzadr[52]
rectangle at (205,435)-(236,466): text "52"; invisible if not DALI_Config.Kurzadr[52]; alarm colour if DALI_Config.Lampenausfall[52]
rectangle at (245,435)-(276,466): text "53"; alarm colour if DALI_Config.Kurzadr[53]
rectangle at (245,435)-(276,466): text "53"; invisible if not DALI_Config.Kurzadr[53]; alarm colour if DALI_Config.Lampenausfall[53]
rectangle at (285,435)-(316,466): text "54"; alarm colour if DALI_Config.Kurzadr[54]
rectangle at (285,435)-(316,466): text "54"; invisible if not DALI_Config.Kurzadr[54]; alarm colour if DALI_Config.Lampenausfall[54]
rectangle at (325,435)-(356,466): text "55"; alarm colour if DALI_Config.Kurzadr[55]
rectangle at (325,435)-(356,466): text "55"; invisible if not DALI_Config.Kurzadr[55]; alarm colour if DALI_Config.Lampenausfall[55]
rectangle at (365,435)-(396,466): text "56"; alarm colour if DALI_Config.Kurzadr[56]
rectangle at (365,435)-(396,466): text "56"; invisible if not DALI_Config.Kurzadr[56]; alarm colour if DALI_Config.Lampenausfall[56]
rectangle at (405,435)-(436,466): text "57"; alarm colour if DALI_Config.Kurzadr[57]
rectangle at (405,435)-(436,466): text "57"; invisible if not DALI_Config.Kurzadr[57]; alarm colour if DALI_Config.Lampenausfall[57]
rectangle at (485,435)-(516,466): text "59"; alarm colour if DALI_Config.Kurzadr[59]
rectangle at (485,435)-(516,466): text "59"; invisible if not DALI_Config.Kurzadr[59]; alarm colour if DALI_Config.Lampenausfall[59]
rectangle at (525,435)-(556,466): text "60"; alarm colour if DALI_Config.Kurzadr[60]
rectangle at (525,435)-(556,466): text "60"; invisible if not DALI_Config.Kurzadr[60]; alarm colour if DALI_Config.Lampenausfall[60]
rectangle at (565,435)-(596,466): text "61"; alarm colour if DALI_Config.Kurzadr[61]
rectangle at (565,435)-(596,466): text "61"; invisible if not DALI_Config.Kurzadr[61]; alarm colour if DALI_Config.Lampenausfall[61]
rectangle at (605,435)-(636,466): text "62"; alarm colour if DALI_Config.Kurzadr[62]
rectangle at (605,435)-(636,466): text "62"; invisible if not DALI_Config.Kurzadr[62]; alarm colour if DALI_Config.Lampenausfall[62]
rectangle at (445,435)-(476,466): text "58"; alarm colour if DALI_Config.Kurzadr[58]
rectangle at (445,435)-(476,466): text "58"; invisible if not DALI_Config.Kurzadr[58]; alarm colour if DALI_Config.Lampenausfall[58]
rectangle at (645,435)-(676,466): text "63"; alarm colour if DALI_Config.Kurzadr[63]
rectangle at (645,435)-(676,466): text "63"; invisible if not DALI_Config.Kurzadr[63]; alarm colour if DALI_Config.Lampenausfall[63]
rectangle at (685,435)-(716,466): text "64"; alarm colour if DALI_Config.Kurzadr[64]
rectangle at (685,435)-(716,466): text "64"; invisible if not DALI_Config.Kurzadr[64]; alarm colour if DALI_Config.Lampenausfall[64]
button at (325,485)-(476,521): text "Query status"; taps DALI_Config.Status; tooltip If you click the button "Query Status", you will get the status "Lamp failure" and "Lamp arc power on" from the ECG.
rectangle at (90,485)-(251,506): text "Short address available"
rectangle at (105,515)-(236,536): text "Lamp failure"
rectangle at (105,545)-(176,566): text "Lamp on"
6 more shapes without text or variables
*)

(* Visualisation PLC_VISU
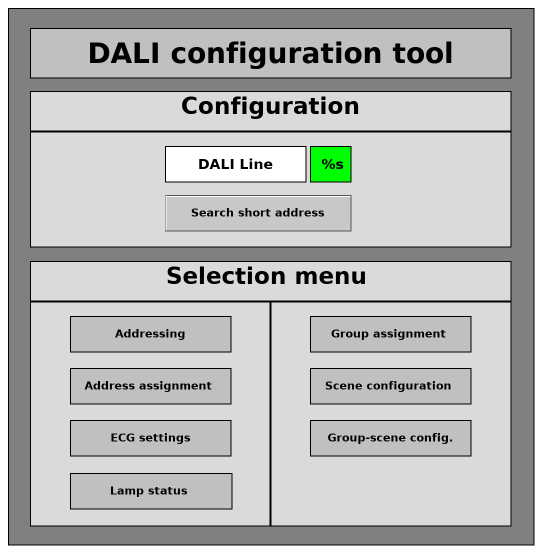
rectangle at (171,91)-(652,247): text "Configuration"
rectangle at (171,261)-(652,526): text "Selection menu"
rectangle at (171,28)-(652,78): text "DALI configuration tool"
rectangle at (211,316)-(372,352): text "Addressing"; opens Addressing
rectangle at (211,368)-(372,404): text "Address assignment"; opens Sort_short_address
rectangle at (451,316)-(612,352): text "Group assignment"; opens group_assignment
rectangle at (451,368)-(612,404): text "Scene configuration"; opens Scene_configuration
rectangle at (211,420)-(372,456): text "ECG settings"; opens ECG_settings
rectangle at (451,420)-(612,456): text "Group-scene config."; opens GroupSceneConfiguration
rectangle at (306,146)-(447,182): text "DALI Line"
button at (306,195)-(492,231): text "Search short address"; taps DALI_Config.SucheKurzadr; tooltip Clicking the button "Search Short Address" will start the search for available short addresses.
rectangle at (451,146)-(492,182): text "%s"; shows DALI_Config.Dali_Linie; alarm colour if DALI_Config.keineJobliste; tooltip Select DALI Line (1 - 5); editable
rectangle at (211,473)-(373,509): text "Lamp status"; opens Lamp_status
4 more shapes without text or variables
*)

(* Visualisation Scene_configuration
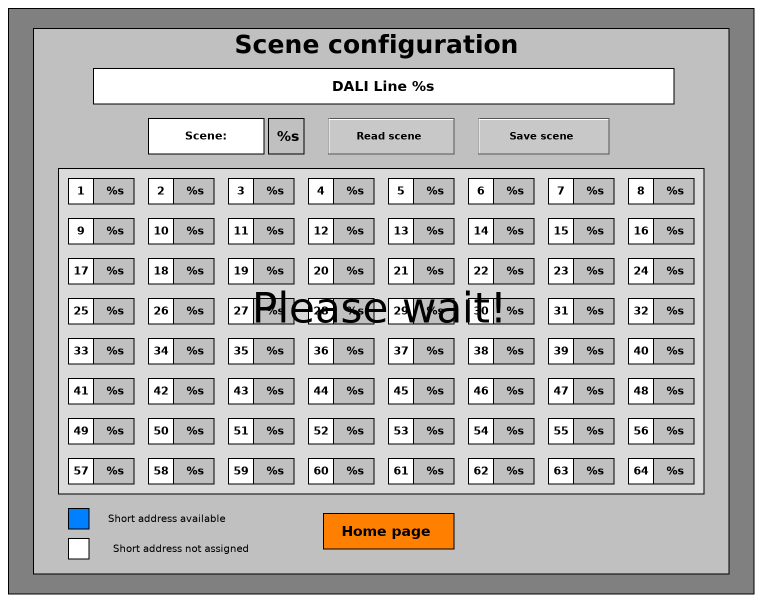
rectangle at (50,25)-(746,571): text "Scene configuration"
rounded rectangle at (340,510)-(471,546): text "Home page"; opens PLC_VISU; tooltip Back to home page
rounded rectangle at (110,65)-(691,101): text "DALI Line %s"; shows DALI_Config.bDali_Linie; tooltip You can change the DALI Line only on the home page.
rectangle at (85,175)-(111,201): text "1"; alarm colour if Dali_Config.Kurzadr[1]
rectangle at (110,175)-(151,201): text "%s"; shows DALI_Config.Szenenwert[1]; tooltip 0 % = Off 1 - 100 % = Dim level 101 % = Mask; editable
button at (495,115)-(626,151): text "Save scene"; taps DALI_Config.SzeneSpeichern; tooltip Save the configured dim levels in the ECGs.
button at (345,115)-(471,151): text "Read scene"; taps DALI_Config.SzeneLesen; tooltip Read the saved scene values from the ECGs.
rectangle at (85,215)-(111,241): text "9"; alarm colour if Dali_Config.Kurzadr[9]
rectangle at (110,215)-(151,241): text "%s"; shows DALI_Config.Szenenwert[9]; tooltip 0 % = Off 1 - 100 % = Dim level 101 % = Mask; editable
rectangle at (85,255)-(111,281): text "17"; alarm colour if Dali_Config.Kurzadr[17]
rectangle at (110,255)-(151,281): text "%s"; shows DALI_Config.Szenenwert[17]; tooltip 0 % = Off 1 - 100 % = Dim level 101 % = Mask; editable
rectangle at (85,295)-(111,321): text "25"; alarm colour if Dali_Config.Kurzadr[25]
rectangle at (110,295)-(151,321): text "%s"; shows DALI_Config.Szenenwert[25]; tooltip 0 % = Off 1 - 100 % = Dim level 101 % = Mask; editable
rectangle at (85,335)-(111,361): text "33"; alarm colour if Dali_Config.Kurzadr[33]
rectangle at (110,335)-(151,361): text "%s"; shows DALI_Config.Szenenwert[33]; tooltip 0 % = Off 1 - 100 % = Dim level 101 % = Mask; editable
rectangle at (85,375)-(111,401): text "41"; alarm colour if Dali_Config.Kurzadr[41]
rectangle at (110,375)-(151,401): text "%s"; shows DALI_Config.Szenenwert[41]; tooltip 0 % = Off 1 - 100 % = Dim level 101 % = Mask; editable
rectangle at (85,415)-(111,441): text "49"; alarm colour if Dali_Config.Kurzadr[49]
rectangle at (110,415)-(151,441): text "%s"; shows DALI_Config.Szenenwert[49]; tooltip 0 % = Off 1 - 100 % = Dim level 101 % = Mask; editable
rectangle at (85,455)-(111,481): text "57"; alarm colour if Dali_Config.Kurzadr[57]
rectangle at (110,455)-(151,481): text "%s"; shows DALI_Config.Szenenwert[57]; tooltip 0 % = Off 1 - 100 % = Dim level 101 % = Mask; editable
rectangle at (165,175)-(191,201): text "2"; alarm colour if Dali_Config.Kurzadr[2]
rectangle at (190,175)-(231,201): text "%s"; shows DALI_Config.Szenenwert[2]; tooltip 0 % = Off 1 - 100 % = Dim level 101 % = Mask; editable
rectangle at (165,215)-(191,241): text "10"; alarm colour if Dali_Config.Kurzadr[10]
rectangle at (190,215)-(231,241): text "%s"; shows DALI_Config.Szenenwert[10]; tooltip 0 % = Off 1 - 100 % = Dim level 101 % = Mask; editable
rectangle at (165,255)-(191,281): text "18"; alarm colour if Dali_Config.Kurzadr[18]
rectangle at (190,255)-(231,281): text "%s"; shows DALI_Config.Szenenwert[18]; tooltip 0 % = Off 1 - 100 % = Dim level 101 % = Mask; editable
rectangle at (165,295)-(191,321): text "26"; alarm colour if Dali_Config.Kurzadr[26]
rectangle at (190,295)-(231,321): text "%s"; shows DALI_Config.Szenenwert[26]; tooltip 0 % = Off 1 - 100 % = Dim level 101 % = Mask; editable
rectangle at (165,335)-(191,361): text "34"; alarm colour if Dali_Config.Kurzadr[34]
rectangle at (190,335)-(231,361): text "%s"; shows DALI_Config.Szenenwert[34]; tooltip 0 % = Off 1 - 100 % = Dim level 101 % = Mask; editable
rectangle at (165,375)-(191,401): text "42"; alarm colour if Dali_Config.Kurzadr[42]
rectangle at (190,375)-(231,401): text "%s"; shows DALI_Config.Szenenwert[42]; tooltip 0 % = Off 1 - 100 % = Dim level 101 % = Mask; editable
rectangle at (165,415)-(191,441): text "50"; alarm colour if Dali_Config.Kurzadr[50]
rectangle at (190,415)-(231,441): text "%s"; shows DALI_Config.Szenenwert[50]; tooltip 0 % = Off 1 - 100 % = Dim level 101 % = Mask; editable
rectangle at (165,455)-(191,481): text "58"; alarm colour if Dali_Config.Kurzadr[58]
rectangle at (190,455)-(231,481): text "%s"; shows DALI_Config.Szenenwert[58]; tooltip 0 % = Off 1 - 100 % = Dim level 101 % = Mask; editable
rectangle at (245,175)-(271,201): text "3"; alarm colour if Dali_Config.Kurzadr[3]
rectangle at (270,175)-(311,201): text "%s"; shows DALI_Config.Szenenwert[3]; tooltip 0 % = Off 1 - 100 % = Dim level 101 % = Mask; editable
rectangle at (245,215)-(271,241): text "11"; alarm colour if Dali_Config.Kurzadr[11]
rectangle at (270,215)-(311,241): text "%s"; shows DALI_Config.Szenenwert[11]; tooltip 0 % = Off 1 - 100 % = Dim level 101 % = Mask; editable
rectangle at (245,255)-(271,281): text "19"; alarm colour if Dali_Config.Kurzadr[19]
rectangle at (270,255)-(311,281): text "%s"; shows DALI_Config.Szenenwert[19]; tooltip 0 % = Off 1 - 100 % = Dim level 101 % = Mask; editable
rectangle at (245,295)-(271,321): text "27"; alarm colour if Dali_Config.Kurzadr[27]
rectangle at (270,295)-(311,321): text "%s"; shows DALI_Config.Szenenwert[27]; tooltip 0 % = Off 1 - 100 % = Dim level 101 % = Mask; editable
rectangle at (245,335)-(271,361): text "35"; alarm colour if Dali_Config.Kurzadr[35]
rectangle at (270,335)-(311,361): text "%s"; shows DALI_Config.Szenenwert[35]; tooltip 0 % = Off 1 - 100 % = Dim level 101 % = Mask; editable
rectangle at (245,375)-(271,401): text "43"; alarm colour if Dali_Config.Kurzadr[43]
rectangle at (270,375)-(311,401): text "%s"; shows DALI_Config.Szenenwert[43]; tooltip 0 % = Off 1 - 100 % = Dim level 101 % = Mask; editable
rectangle at (245,415)-(271,441): text "51"; alarm colour if Dali_Config.Kurzadr[51]
rectangle at (270,415)-(311,441): text "%s"; shows DALI_Config.Szenenwert[51]; tooltip 0 % = Off 1 - 100 % = Dim level 101 % = Mask; editable
rectangle at (245,455)-(271,481): text "59"; alarm colour if Dali_Config.Kurzadr[59]
rectangle at (270,455)-(311,481): text "%s"; shows DALI_Config.Szenenwert[59]; tooltip 0 % = Off 1 - 100 % = Dim level 101 % = Mask; editable
rectangle at (325,175)-(351,201): text "4"; alarm colour if Dali_Config.Kurzadr[4]
rectangle at (350,175)-(391,201): text "%s"; shows DALI_Config.Szenenwert[4]; tooltip 0 % = Off 1 - 100 % = Dim level 101 % = Mask; editable
rectangle at (325,215)-(351,241): text "12"; alarm colour if Dali_Config.Kurzadr[12]
rectangle at (350,215)-(391,241): text "%s"; shows DALI_Config.Szenenwert[12]; tooltip 0 % = Off 1 - 100 % = Dim level 101 % = Mask; editable
rectangle at (325,255)-(351,281): text "20"; alarm colour if Dali_Config.Kurzadr[20]
rectangle at (350,255)-(391,281): text "%s"; shows DALI_Config.Szenenwert[20]; tooltip 0 % = Off 1 - 100 % = Dim level 101 % = Mask; editable
rectangle at (325,295)-(351,321): text "28"; alarm colour if Dali_Config.Kurzadr[28]
rectangle at (350,295)-(391,321): text "%s"; shows DALI_Config.Szenenwert[28]; tooltip 0 % = Off 1 - 100 % = Dim level 101 % = Mask; editable
rectangle at (325,335)-(351,361): text "36"; alarm colour if Dali_Config.Kurzadr[36]
rectangle at (350,335)-(391,361): text "%s"; shows DALI_Config.Szenenwert[36]; tooltip 0 % = Off 1 - 100 % = Dim level 101 % = Mask; editable
rectangle at (325,375)-(351,401): text "44"; alarm colour if Dali_Config.Kurzadr[44]
rectangle at (350,375)-(391,401): text "%s"; shows DALI_Config.Szenenwert[44]; tooltip 0 % = Off 1 - 100 % = Dim level 101 % = Mask; editable
rectangle at (325,415)-(351,441): text "52"; alarm colour if Dali_Config.Kurzadr[52]
rectangle at (350,415)-(391,441): text "%s"; shows DALI_Config.Szenenwert[52]; tooltip 0 % = Off 1 - 100 % = Dim level 101 % = Mask; editable
rectangle at (325,455)-(351,481): text "60"; alarm colour if Dali_Config.Kurzadr[60]
rectangle at (350,455)-(391,481): text "%s"; shows DALI_Config.Szenenwert[60]; tooltip 0 % = Off 1 - 100 % = Dim level 101 % = Mask; editable
rectangle at (405,175)-(431,201): text "5"; alarm colour if Dali_Config.Kurzadr[5]
rectangle at (430,175)-(471,201): text "%s"; shows DALI_Config.Szenenwert[5]; tooltip 0 % = Off 1 - 100 % = Dim level 101 % = Mask; editable
rectangle at (405,215)-(431,241): text "13"; alarm colour if Dali_Config.Kurzadr[13]
rectangle at (430,215)-(471,241): text "%s"; shows DALI_Config.Szenenwert[13]; tooltip 0 % = Off 1 - 100 % = Dim level 101 % = Mask; editable
rectangle at (405,255)-(431,281): text "21"; alarm colour if Dali_Config.Kurzadr[21]
rectangle at (430,255)-(471,281): text "%s"; shows DALI_Config.Szenenwert[21]; tooltip 0 % = Off 1 - 100 % = Dim level 101 % = Mask; editable
rectangle at (405,295)-(431,321): text "29"; alarm colour if Dali_Config.Kurzadr[29]
rectangle at (430,295)-(471,321): text "%s"; shows DALI_Config.Szenenwert[29]; tooltip 0 % = Off 1 - 100 % = Dim level 101 % = Mask; editable
rectangle at (405,335)-(431,361): text "37"; alarm colour if Dali_Config.Kurzadr[37]
rectangle at (430,335)-(471,361): text "%s"; shows DALI_Config.Szenenwert[37]; tooltip 0 % = Off 1 - 100 % = Dim level 101 % = Mask; editable
rectangle at (405,375)-(431,401): text "45"; alarm colour if Dali_Config.Kurzadr[45]
rectangle at (430,375)-(471,401): text "%s"; shows DALI_Config.Szenenwert[45]; tooltip 0 % = Off 1 - 100 % = Dim level 101 % = Mask; editable
rectangle at (405,415)-(431,441): text "53"; alarm colour if Dali_Config.Kurzadr[53]
rectangle at (430,415)-(471,441): text "%s"; shows DALI_Config.Szenenwert[53]; tooltip 0 % = Off 1 - 100 % = Dim level 101 % = Mask; editable
rectangle at (405,455)-(431,481): text "61"; alarm colour if Dali_Config.Kurzadr[61]
rectangle at (430,455)-(471,481): text "%s"; shows DALI_Config.Szenenwert[61]; tooltip 0 % = Off 1 - 100 % = Dim level 101 % = Mask; editable
rectangle at (485,175)-(511,201): text "6"; alarm colour if Dali_Config.Kurzadr[6]
rectangle at (510,175)-(551,201): text "%s"; shows DALI_Config.Szenenwert[6]; tooltip 0 % = Off 1 - 100 % = Dim level 101 % = Mask; editable
rectangle at (485,215)-(511,241): text "14"; alarm colour if Dali_Config.Kurzadr[14]
rectangle at (510,215)-(551,241): text "%s"; shows DALI_Config.Szenenwert[14]; tooltip 0 % = Off 1 - 100 % = Dim level 101 % = Mask; editable
rectangle at (485,255)-(511,281): text "22"; alarm colour if Dali_Config.Kurzadr[22]
rectangle at (510,255)-(551,281): text "%s"; shows DALI_Config.Szenenwert[22]; tooltip 0 % = Off 1 - 100 % = Dim level 101 % = Mask; editable
rectangle at (485,295)-(511,321): text "30"; alarm colour if Dali_Config.Kurzadr[30]
rectangle at (510,295)-(551,321): text "%s"; shows DALI_Config.Szenenwert[30]; tooltip 0 % = Off 1 - 100 % = Dim level 101 % = Mask; editable
rectangle at (485,335)-(511,361): text "38"; alarm colour if Dali_Config.Kurzadr[38]
rectangle at (510,335)-(551,361): text "%s"; shows DALI_Config.Szenenwert[38]; tooltip 0 % = Off 1 - 100 % = Dim level 101 % = Mask; editable
rectangle at (485,375)-(511,401): text "46"; alarm colour if Dali_Config.Kurzadr[46]
rectangle at (510,375)-(551,401): text "%s"; shows DALI_Config.Szenenwert[46]; tooltip 0 % = Off 1 - 100 % = Dim level 101 % = Mask; editable
rectangle at (485,415)-(511,441): text "54"; alarm colour if Dali_Config.Kurzadr[54]
rectangle at (510,415)-(551,441): text "%s"; shows DALI_Config.Szenenwert[54]; tooltip 0 % = Off 1 - 100 % = Dim level 101 % = Mask; editable
rectangle at (485,455)-(511,481): text "62"; alarm colour if Dali_Config.Kurzadr[62]
rectangle at (510,455)-(551,481): text "%s"; shows DALI_Config.Szenenwert[62]; tooltip 0 % = Off 1 - 100 % = Dim level 101 % = Mask; editable
rectangle at (565,175)-(591,201): text "7"; alarm colour if Dali_Config.Kurzadr[7]
rectangle at (590,175)-(631,201): text "%s"; shows DALI_Config.Szenenwert[7]; tooltip 0 % = Off 1 - 100 % = Dim level 101 % = Mask; editable
rectangle at (565,215)-(591,241): text "15"; alarm colour if Dali_Config.Kurzadr[15]
rectangle at (590,215)-(631,241): text "%s"; shows DALI_Config.Szenenwert[15]; tooltip 0 % = Off 1 - 100 % = Dim level 101 % = Mask; editable
rectangle at (565,255)-(591,281): text "23"; alarm colour if Dali_Config.Kurzadr[23]
rectangle at (590,255)-(631,281): text "%s"; shows DALI_Config.Szenenwert[23]; tooltip 0 % = Off 1 - 100 % = Dim level 101 % = Mask; editable
rectangle at (565,295)-(591,321): text "31"; alarm colour if Dali_Config.Kurzadr[31]
rectangle at (590,295)-(631,321): text "%s"; shows DALI_Config.Szenenwert[31]; tooltip 0 % = Off 1 - 100 % = Dim level 101 % = Mask; editable
rectangle at (565,335)-(591,361): text "39"; alarm colour if Dali_Config.Kurzadr[39]
rectangle at (590,335)-(631,361): text "%s"; shows DALI_Config.Szenenwert[39]; tooltip 0 % = Off 1 - 100 % = Dim level 101 % = Mask; editable
rectangle at (565,375)-(591,401): text "47"; alarm colour if Dali_Config.Kurzadr[47]
rectangle at (590,375)-(631,401): text "%s"; shows DALI_Config.Szenenwert[47]; tooltip 0 % = Off 1 - 100 % = Dim level 101 % = Mask; editable
rectangle at (565,415)-(591,441): text "55"; alarm colour if Dali_Config.Kurzadr[55]
rectangle at (590,415)-(631,441): text "%s"; shows DALI_Config.Szenenwert[55]; tooltip 0 % = Off 1 - 100 % = Dim level 101 % = Mask; editable
rectangle at (565,455)-(591,481): text "63"; alarm colour if Dali_Config.Kurzadr[63]
rectangle at (590,455)-(631,481): text "%s"; shows DALI_Config.Szenenwert[63]; tooltip 0 % = Off 1 - 100 % = Dim level 101 % = Mask; editable
rectangle at (645,175)-(671,201): text "8"; alarm colour if Dali_Config.Kurzadr[8]
rectangle at (670,175)-(711,201): text "%s"; shows DALI_Config.Szenenwert[8]; tooltip 0 % = Off 1 - 100 % = Dim level 101 % = Mask; editable
rectangle at (645,215)-(671,241): text "16"; alarm colour if Dali_Config.Kurzadr[16]
rectangle at (670,215)-(711,241): text "%s"; shows DALI_Config.Szenenwert[16]; tooltip 0 % = Off 1 - 100 % = Dim level 101 % = Mask; editable
rectangle at (645,255)-(671,281): text "24"; alarm colour if Dali_Config.Kurzadr[24]
rectangle at (670,255)-(711,281): text "%s"; shows DALI_Config.Szenenwert[24]; tooltip 0 % = Off 1 - 100 % = Dim level 101 % = Mask; editable
rectangle at (645,295)-(671,321): text "32"; alarm colour if Dali_Config.Kurzadr[32]
rectangle at (670,295)-(711,321): text "%s"; shows DALI_Config.Szenenwert[32]; tooltip 0 % = Off 1 - 100 % = Dim level 101 % = Mask; editable
rectangle at (645,335)-(671,361): text "40"; alarm colour if Dali_Config.Kurzadr[40]
rectangle at (670,335)-(711,361): text "%s"; shows DALI_Config.Szenenwert[40]; tooltip 0 % = Off 1 - 100 % = Dim level 101 % = Mask; editable
rectangle at (645,375)-(671,401): text "48"; alarm colour if Dali_Config.Kurzadr[48]
rectangle at (670,375)-(711,401): text "%s"; shows DALI_Config.Szenenwert[48]; tooltip 0 % = Off 1 - 100 % = Dim level 101 % = Mask; editable
rectangle at (645,415)-(671,441): text "56"; alarm colour if Dali_Config.Kurzadr[56]
rectangle at (670,415)-(711,441): text "%s"; shows DALI_Config.Szenenwert[56]; tooltip 0 % = Off 1 - 100 % = Dim level 101 % = Mask; editable
rectangle at (645,455)-(671,481): text "64"; alarm colour if Dali_Config.Kurzadr[64]
rectangle at (670,455)-(711,481): text "%s"; shows DALI_Config.Szenenwert[64]; tooltip 0 % = Off 1 - 100 % = Dim level 101 % = Mask; editable
rectangle at (165,115)-(281,151): text "Scene:"
rectangle at (285,115)-(321,151): text "%s"; shows DALI_Config.Szene; tooltip Select scene 1 - 16; editable
rectangle at (110,505)-(261,526): text "Short address available"
rectangle at (105,535)-(291,556): text "Short address not assigned"
rectangle at (51,111)-(742,498): text "Please wait!"; invisible if NOT DALI_Config.Unsichtbar
4 more shapes without text or variables
*)

